# B&R Automation Studio project NAINV104C00R8L515F00 (part 6)

#### fHermesFormBoardAvailable.st
```iecst
(* Hermes Form Board Available Table Data (Total Index Written In Table) *)
FUNCTION fHermesFormBoardAvailable

	memset(ADR(pa_tyXMLTable) , 0 , SIZEOF(pa_tyXMLTable));
	iTotalIdxWrite	:= 0;

	fHermesGetTimestamp(ADR(sTimestamp) , tyDTStructure);

	pa_tyXMLTable[iTotalIdxWrite].sTitle	:= 'ST';
	pa_tyXMLTable[iTotalIdxWrite].sValue	:= 'Hermes';
	pa_tyXMLTable[iTotalIdxWrite].uiSize	:= LEN(pa_tyXMLTable[iTotalIdxWrite].sValue);

	iTotalIdxWrite	:= iTotalIdxWrite + 1;

	pa_tyXMLTable[iTotalIdxWrite].sTitle	:= 'AT';
	pa_tyXMLTable[iTotalIdxWrite].sValue	:= 'Timestamp';
	pa_tyXMLTable[iTotalIdxWrite].uiSize	:= LEN(pa_tyXMLTable[iTotalIdxWrite].sValue);

	iTotalIdxWrite	:= iTotalIdxWrite + 1;

	pa_tyXMLTable[iTotalIdxWrite].sTitle	:= 'AV';
	pa_tyXMLTable[iTotalIdxWrite].sValue	:= sTimestamp;
	pa_tyXMLTable[iTotalIdxWrite].uiSize	:= LEN(pa_tyXMLTable[iTotalIdxWrite].sValue);

	iTotalIdxWrite	:= iTotalIdxWrite + 1;

	pa_tyXMLTable[iTotalIdxWrite].sTitle	:= 'EN';
	pa_tyXMLTable[iTotalIdxWrite].sValue	:= '';
	pa_tyXMLTable[iTotalIdxWrite].uiSize	:= LEN(pa_tyXMLTable[iTotalIdxWrite].sValue);

	iTotalIdxWrite	:= iTotalIdxWrite + 1;

	pa_tyXMLTable[iTotalIdxWrite].sTitle	:= 'ST';
	pa_tyXMLTable[iTotalIdxWrite].sValue	:= 'BoardAvailable';
	pa_tyXMLTable[iTotalIdxWrite].uiSize	:= LEN(pa_tyXMLTable[iTotalIdxWrite].sValue);

	iTotalIdxWrite	:= iTotalIdxWrite + 1;

	IF tyParameter.tyAvl.bBoardId = TRUE THEN
		pa_tyXMLTable[iTotalIdxWrite].sTitle	:= 'AT';
		pa_tyXMLTable[iTotalIdxWrite].sValue	:= 'BoardId';
		pa_tyXMLTable[iTotalIdxWrite].uiSize	:= LEN(pa_tyXMLTable[iTotalIdxWrite].sValue);

		iTotalIdxWrite	:= iTotalIdxWrite + 1;

		pa_tyXMLTable[iTotalIdxWrite].sTitle	:= 'AV';
		pa_tyXMLTable[iTotalIdxWrite].sValue	:= tyParameter.tyData.sBoardId;
		pa_tyXMLTable[iTotalIdxWrite].uiSize	:= LEN(pa_tyXMLTable[iTotalIdxWrite].sValue);

		iTotalIdxWrite	:= iTotalIdxWrite + 1;
	END_IF

	IF tyParameter.tyAvl.bBoardIdCreatedBy = TRUE THEN
		pa_tyXMLTable[iTotalIdxWrite].sTitle	:= 'AT';
		pa_tyXMLTable[iTotalIdxWrite].sValue	:= 'BoardIdCreatedBy';
		pa_tyXMLTable[iTotalIdxWrite].uiSize	:= LEN(pa_tyXMLTable[iTotalIdxWrite].sValue);

		iTotalIdxWrite	:= iTotalIdxWrite + 1;

		pa_tyXMLTable[iTotalIdxWrite].sTitle	:= 'AV';
		pa_tyXMLTable[iTotalIdxWrite].sValue	:= tyParameter.tyData.sBoardIdCreatedBy;
		pa_tyXMLTable[iTotalIdxWrite].uiSize	:= LEN(pa_tyXMLTable[iTotalIdxWrite].sValue);

		iTotalIdxWrite	:= iTotalIdxWrite + 1;
	END_IF

	IF tyParameter.tyAvl.bFailedBoard = TRUE THEN
		pa_tyXMLTable[iTotalIdxWrite].sTitle	:= 'AT';
		pa_tyXMLTable[iTotalIdxWrite].sValue	:= 'FailedBoard';
		pa_tyXMLTable[iTotalIdxWrite].uiSize	:= LEN(pa_tyXMLTable[iTotalIdxWrite].sValue);

		iTotalIdxWrite	:= iTotalIdxWrite + 1;

		pa_tyXMLTable[iTotalIdxWrite].sTitle	:= 'AV';
		pa_tyXMLTable[iTotalIdxWrite].sValue	:= DINT_TO_STRING(UDINT_TO_DINT(tyParameter.tyData.eFailedBoard));
		pa_tyXMLTable[iTotalIdxWrite].uiSize	:= LEN(pa_tyXMLTable[iTotalIdxWrite].sValue);

		iTotalIdxWrite	:= iTotalIdxWrite + 1;
	END_IF

	IF tyParameter.tyAvl.bProductTypeId = TRUE THEN
		pa_tyXMLTable[iTotalIdxWrite].sTitle	:= 'AT';
		pa_tyXMLTable[iTotalIdxWrite].sValue	:= 'ProductTypeId';
		pa_tyXMLTable[iTotalIdxWrite].uiSize	:= LEN(pa_tyXMLTable[iTotalIdxWrite].sValue);

		iTotalIdxWrite	:= iTotalIdxWrite + 1;

		pa_tyXMLTable[iTotalIdxWrite].sTitle	:= 'AV';
		pa_tyXMLTable[iTotalIdxWrite].sValue	:= tyParameter.tyData.sProductTypeId;
		pa_tyXMLTable[iTotalIdxWrite].uiSize	:= LEN(pa_tyXMLTable[iTotalIdxWrite].sValue);

		iTotalIdxWrite	:= iTotalIdxWrite + 1;
	END_IF

	IF tyParameter.tyAvl.bFlippedBoard = TRUE THEN
		pa_tyXMLTable[iTotalIdxWrite].sTitle	:= 'AT';
		pa_tyXMLTable[iTotalIdxWrite].sValue	:= 'FlippedBoard';
		pa_tyXMLTable[iTotalIdxWrite].uiSize	:= LEN(pa_tyXMLTable[iTotalIdxWrite].sValue);

		iTotalIdxWrite	:= iTotalIdxWrite + 1;

		pa_tyXMLTable[iTotalIdxWrite].sTitle	:= 'AV';
		pa_tyXMLTable[iTotalIdxWrite].sValue	:= DINT_TO_STRING(UDINT_TO_DINT(tyParameter.tyData.eFlippedBoard));
		pa_tyXMLTable[iTotalIdxWrite].uiSize	:= LEN(pa_tyXMLTable[iTotalIdxWrite].sValue);

		iTotalIdxWrite	:= iTotalIdxWrite + 1;
	END_IF

	IF tyParameter.tyAvl.bTopBarcode = TRUE THEN
		pa_tyXMLTable[iTotalIdxWrite].sTitle	:= 'AT';
		pa_tyXMLTable[iTotalIdxWrite].sValue	:= 'TopBarcode';
		pa_tyXMLTable[iTotalIdxWrite].uiSize	:= LEN(pa_tyXMLTable[iTotalIdxWrite].sValue);

		iTotalIdxWrite	:= iTotalIdxWrite + 1;

		pa_tyXMLTable[iTotalIdxWrite].sTitle	:= 'AV';
		pa_tyXMLTable[iTotalIdxWrite].sValue	:= tyParameter.tyData.sTopBarcode;
		pa_tyXMLTable[iTotalIdxWrite].uiSize	:= LEN(pa_tyXMLTable[iTotalIdxWrite].sValue);

		iTotalIdxWrite	:= iTotalIdxWrite + 1;
	END_IF

	IF tyParameter.tyAvl.bBottomBarcode = TRUE THEN
		pa_tyXMLTable[iTotalIdxWrite].sTitle	:= 'AT';
		pa_tyXMLTable[iTotalIdxWrite].sValue	:= 'BottomBarcode';
		pa_tyXMLTable[iTotalIdxWrite].uiSize	:= LEN(pa_tyXMLTable[iTotalIdxWrite].sValue);

		iTotalIdxWrite	:= iTotalIdxWrite + 1;

		pa_tyXMLTable[iTotalIdxWrite].sTitle	:= 'AV';
		pa_tyXMLTable[iTotalIdxWrite].sValue	:= tyParameter.tyData.sBottomBarcode;
		pa_tyXMLTable[iTotalIdxWrite].uiSize	:= LEN(pa_tyXMLTable[iTotalIdxWrite].sValue);

		iTotalIdxWrite	:= iTotalIdxWrite + 1;
	END_IF

	IF tyParameter.tyAvl.bLength = TRUE THEN
		pa_tyXMLTable[iTotalIdxWrite].sTitle	:= 'AT';
		pa_tyXMLTable[iTotalIdxWrite].sValue	:= 'Length';
		pa_tyXMLTable[iTotalIdxWrite].uiSize	:= LEN(pa_tyXMLTable[iTotalIdxWrite].sValue);

		iTotalIdxWrite	:= iTotalIdxWrite + 1;

		pa_tyXMLTable[iTotalIdxWrite].sTitle	:= 'AV';
		pa_tyXMLTable[iTotalIdxWrite].sValue	:= REAL_TO_STRING(tyParameter.tyData.rLength);
		pa_tyXMLTable[iTotalIdxWrite].uiSize	:= LEN(pa_tyXMLTable[iTotalIdxWrite].sValue);

		iTotalIdxWrite	:= iTotalIdxWrite + 1;
	END_IF

	IF tyParameter.tyAvl.bWidth = TRUE THEN
		pa_tyXMLTable[iTotalIdxWrite].sTitle	:= 'AT';
		pa_tyXMLTable[iTotalIdxWrite].sValue	:= 'Width';
		pa_tyXMLTable[iTotalIdxWrite].uiSize	:= LEN(pa_tyXMLTable[iTotalIdxWrite].sValue);

		iTotalIdxWrite	:= iTotalIdxWrite + 1;

		pa_tyXMLTable[iTotalIdxWrite].sTitle	:= 'AV';
		pa_tyXMLTable[iTotalIdxWrite].sValue	:= REAL_TO_STRING(tyParameter.tyData.rWidth);
		pa_tyXMLTable[iTotalIdxWrite].uiSize	:= LEN(pa_tyXMLTable[iTotalIdxWrite].sValue);

		iTotalIdxWrite	:= iTotalIdxWrite + 1;
	END_IF

	IF tyParameter.tyAvl.bThickness = TRUE THEN
		pa_tyXMLTable[iTotalIdxWrite].sTitle	:= 'AT';
		pa_tyXMLTable[iTotalIdxWrite].sValue	:= 'Thickness';
		pa_tyXMLTable[iTotalIdxWrite].uiSize	:= LEN(pa_tyXMLTable[iTotalIdxWrite].sValue);

		iTotalIdxWrite	:= iTotalIdxWrite + 1;

		pa_tyXMLTable[iTotalIdxWrite].sTitle	:= 'AV';
		pa_tyXMLTable[iTotalIdxWrite].sValue	:= REAL_TO_STRING(tyParameter.tyData.rThickness);
		pa_tyXMLTable[iTotalIdxWrite].uiSize	:= LEN(pa_tyXMLTable[iTotalIdxWrite].sValue);

		iTotalIdxWrite	:= iTotalIdxWrite + 1;
	END_IF

	IF tyParameter.tyAvl.bConveyorSpeed = TRUE THEN
		pa_tyXMLTable[iTotalIdxWrite].sTitle	:= 'AT';
		pa_tyXMLTable[iTotalIdxWrite].sValue	:= 'ConveyorSpeed';
		pa_tyXMLTable[iTotalIdxWrite].uiSize	:= LEN(pa_tyXMLTable[iTotalIdxWrite].sValue);

		iTotalIdxWrite	:= iTotalIdxWrite + 1;

		pa_tyXMLTable[iTotalIdxWrite].sTitle	:= 'AV';
		pa_tyXMLTable[iTotalIdxWrite].sValue	:= REAL_TO_STRING(tyParameter.tyData.rConveyorSpeed);
		pa_tyXMLTable[iTotalIdxWrite].uiSize	:= LEN(pa_tyXMLTable[iTotalIdxWrite].sValue);

		iTotalIdxWrite	:= iTotalIdxWrite + 1;
	END_IF

	IF tyParameter.tyAvl.bTopClearanceHeight = TRUE THEN
		pa_tyXMLTable[iTotalIdxWrite].sTitle	:= 'AT';
		pa_tyXMLTable[iTotalIdxWrite].sValue	:= 'TopClearanceHeight';
		pa_tyXMLTable[iTotalIdxWrite].uiSize	:= LEN(pa_tyXMLTable[iTotalIdxWrite].sValue);

		iTotalIdxWrite	:= iTotalIdxWrite + 1;

		pa_tyXMLTable[iTotalIdxWrite].sTitle	:= 'AV';
		pa_tyXMLTable[iTotalIdxWrite].sValue	:= REAL_TO_STRING(tyParameter.tyData.rTopClearanceHeight);
		pa_tyXMLTable[iTotalIdxWrite].uiSize	:= LEN(pa_tyXMLTable[iTotalIdxWrite].sValue);

		iTotalIdxWrite	:= iTotalIdxWrite + 1;
	END_IF

	IF tyParameter.tyAvl.bBottomClearanceHeight = TRUE THEN
		pa_tyXMLTable[iTotalIdxWrite].sTitle	:= 'AT';
		pa_tyXMLTable[iTotalIdxWrite].sValue	:= 'BottomClearanceHeight';
		pa_tyXMLTable[iTotalIdxWrite].uiSize	:= LEN(pa_tyXMLTable[iTotalIdxWrite].sValue);

		iTotalIdxWrite	:= iTotalIdxWrite + 1;

		pa_tyXMLTable[iTotalIdxWrite].sTitle	:= 'AV';
		pa_tyXMLTable[iTotalIdxWrite].sValue	:= REAL_TO_STRING(tyParameter.tyData.rBottomClearanceHeight);
		pa_tyXMLTable[iTotalIdxWrite].uiSize	:= LEN(pa_tyXMLTable[iTotalIdxWrite].sValue);

		iTotalIdxWrite	:= iTotalIdxWrite + 1;
	END_IF

	IF tyParameter.tyAvl.bWeight = TRUE THEN
		pa_tyXMLTable[iTotalIdxWrite].sTitle	:= 'AT';
		pa_tyXMLTable[iTotalIdxWrite].sValue	:= 'Weight';
		pa_tyXMLTable[iTotalIdxWrite].uiSize	:= LEN(pa_tyXMLTable[iTotalIdxWrite].sValue);

		iTotalIdxWrite	:= iTotalIdxWrite + 1;

		pa_tyXMLTable[iTotalIdxWrite].sTitle	:= 'AV';
		pa_tyXMLTable[iTotalIdxWrite].sValue	:= REAL_TO_STRING(tyParameter.tyData.rWeight);
		pa_tyXMLTable[iTotalIdxWrite].uiSize	:= LEN(pa_tyXMLTable[iTotalIdxWrite].sValue);

		iTotalIdxWrite	:= iTotalIdxWrite + 1;
	END_IF

	IF tyParameter.tyAvl.bWorkOrderId = TRUE THEN
		pa_tyXMLTable[iTotalIdxWrite].sTitle	:= 'AT';
		pa_tyXMLTable[iTotalIdxWrite].sValue	:= 'WorkOrderId';
		pa_tyXMLTable[iTotalIdxWrite].uiSize	:= LEN(pa_tyXMLTable[iTotalIdxWrite].sValue);

		iTotalIdxWrite	:= iTotalIdxWrite + 1;

		pa_tyXMLTable[iTotalIdxWrite].sTitle	:= 'AV';
		pa_tyXMLTable[iTotalIdxWrite].sValue	:= tyParameter.tyData.sWorkOrderId;
		pa_tyXMLTable[iTotalIdxWrite].uiSize	:= LEN(pa_tyXMLTable[iTotalIdxWrite].sValue);

		iTotalIdxWrite	:= iTotalIdxWrite + 1;
	END_IF

	IF tyParameter.tyAvl.bBatchId = TRUE THEN
		pa_tyXMLTable[iTotalIdxWrite].sTitle	:= 'AT';
		pa_tyXMLTable[iTotalIdxWrite].sValue	:= 'BatchId';
		pa_tyXMLTable[iTotalIdxWrite].uiSize	:= LEN(pa_tyXMLTable[iTotalIdxWrite].sValue);

		iTotalIdxWrite	:= iTotalIdxWrite + 1;

		pa_tyXMLTable[iTotalIdxWrite].sTitle	:= 'AV';
		pa_tyXMLTable[iTotalIdxWrite].sValue	:= tyParameter.tyData.sBatchId;
		pa_tyXMLTable[iTotalIdxWrite].uiSize	:= LEN(pa_tyXMLTable[iTotalIdxWrite].sValue);

		iTotalIdxWrite	:= iTotalIdxWrite + 1;
	END_IF

	IF tyParameter.tyAvl.bRoute = TRUE THEN
		pa_tyXMLTable[iTotalIdxWrite].sTitle	:= 'AT';
		pa_tyXMLTable[iTotalIdxWrite].sValue	:= 'Route';
		pa_tyXMLTable[iTotalIdxWrite].uiSize	:= LEN(pa_tyXMLTable[iTotalIdxWrite].sValue);

		iTotalIdxWrite	:= iTotalIdxWrite + 1;

		pa_tyXMLTable[iTotalIdxWrite].sTitle	:= 'AV';
		pa_tyXMLTable[iTotalIdxWrite].sValue	:= INT_TO_STRING(tyParameter.tyData.iRoute);
		pa_tyXMLTable[iTotalIdxWrite].uiSize	:= LEN(pa_tyXMLTable[iTotalIdxWrite].sValue);

		iTotalIdxWrite	:= iTotalIdxWrite + 1;
	END_IF

	IF tyParameter.tyAvl.bAction = TRUE THEN
		pa_tyXMLTable[iTotalIdxWrite].sTitle	:= 'AT';
		pa_tyXMLTable[iTotalIdxWrite].sValue	:= 'Action';
		pa_tyXMLTable[iTotalIdxWrite].uiSize	:= LEN(pa_tyXMLTable[iTotalIdxWrite].sValue);

		iTotalIdxWrite	:= iTotalIdxWrite + 1;

		pa_tyXMLTable[iTotalIdxWrite].sTitle	:= 'AV';
		pa_tyXMLTable[iTotalIdxWrite].sValue	:= INT_TO_STRING(tyParameter.tyData.iAction);
		pa_tyXMLTable[iTotalIdxWrite].uiSize	:= LEN(pa_tyXMLTable[iTotalIdxWrite].sValue);

		iTotalIdxWrite	:= iTotalIdxWrite + 1;
	END_IF

	//start adding subboard
	IF tyParameter.tyAvl.tySubBoards.bSubBoardsPos[usiSubBoardCntr] <> FALSE OR
		tyParameter.tyAvl.tySubBoards.bSubBoardsBc[usiSubBoardCntr] <> FALSE OR
		tyParameter.tyAvl.tySubBoards.bSubBoardsSt[usiSubBoardCntr] <> FALSE
		THEN
		pa_tyXMLTable[iTotalIdxWrite].sTitle	:= 'EN';
		pa_tyXMLTable[iTotalIdxWrite].sValue	:= '';
		pa_tyXMLTable[iTotalIdxWrite].uiSize	:= LEN(pa_tyXMLTable[iTotalIdxWrite].sValue);

		iTotalIdxWrite	:= iTotalIdxWrite + 1;

		pa_tyXMLTable[iTotalIdxWrite].sTitle	:= 'ST';
		pa_tyXMLTable[iTotalIdxWrite].sValue	:= 'SubBoards';
		pa_tyXMLTable[iTotalIdxWrite].uiSize	:= LEN(pa_tyXMLTable[iTotalIdxWrite].sValue);

		iTotalIdxWrite	:= iTotalIdxWrite + 1;

		pa_tyXMLTable[iTotalIdxWrite].sTitle	:= 'EN';
		pa_tyXMLTable[iTotalIdxWrite].sValue	:= '';
		pa_tyXMLTable[iTotalIdxWrite].uiSize	:= LEN(pa_tyXMLTable[iTotalIdxWrite].sValue);

		iTotalIdxWrite	:= iTotalIdxWrite + 1;

		FOR usiSubBoardCntr := 0  TO SIZEOF(tyParameter.tyAvl.tySubBoards.bSubBoardsPos)/SIZEOF(tyParameter.tyAvl.tySubBoards.bSubBoardsPos[1]) -1 DO
			IF tyParameter.tyAvl.tySubBoards.bSubBoardsPos[usiSubBoardCntr] <> FALSE OR
				tyParameter.tyAvl.tySubBoards.bSubBoardsBc[usiSubBoardCntr] <> FALSE OR
				tyParameter.tyAvl.tySubBoards.bSubBoardsSt[usiSubBoardCntr] <> FALSE
				THEN
				pa_tyXMLTable[iTotalIdxWrite].sTitle	:= 'ST';
				pa_tyXMLTable[iTotalIdxWrite].sValue	:= 'SB';
				pa_tyXMLTable[iTotalIdxWrite].uiSize	:= LEN(pa_tyXMLTable[iTotalIdxWrite].sValue);

				iTotalIdxWrite	:= iTotalIdxWrite + 1;

				pa_tyXMLTable[iTotalIdxWrite].sTitle	:= 'AT';
				pa_tyXMLTable[iTotalIdxWrite].sValue	:= 'Pos';
				pa_tyXMLTable[iTotalIdxWrite].uiSize	:= LEN(pa_tyXMLTable[iTotalIdxWrite].sValue);

				iTotalIdxWrite	:= iTotalIdxWrite + 1;

				pa_tyXMLTable[iTotalIdxWrite].sTitle	:= 'AV';
				pa_tyXMLTable[iTotalIdxWrite].uiSize	:= LEN(pa_tyXMLTable[iTotalIdxWrite].sValue);
				IF tyParameter.tyAvl.tySubBoards.bSubBoardsPos[usiSubBoardCntr] <> FALSE THEN
					pa_tyXMLTable[iTotalIdxWrite].sValue	:= INT_TO_STRING(tyParameter.tyData.tySubBoards.iSubBoardsPos[usiSubBoardCntr]);
				END_IF
				iTotalIdxWrite	:= iTotalIdxWrite + 1;

				pa_tyXMLTable[iTotalIdxWrite].sTitle	:= 'AT';
				pa_tyXMLTable[iTotalIdxWrite].sValue	:= 'Bc';
				pa_tyXMLTable[iTotalIdxWrite].uiSize	:= LEN(pa_tyXMLTable[iTotalIdxWrite].sValue);

				iTotalIdxWrite	:= iTotalIdxWrite + 1;

				pa_tyXMLTable[iTotalIdxWrite].sTitle	:= 'AV';
				IF tyParameter.tyAvl.tySubBoards.bSubBoardsBc[usiSubBoardCntr] <> FALSE THEN
					pa_tyXMLTable[iTotalIdxWrite].sValue	:= tyParameter.tyData.tySubBoards.sSubBoardsBc[usiSubBoardCntr];
				END_IF
				pa_tyXMLTable[iTotalIdxWrite].uiSize	:= LEN(pa_tyXMLTable[iTotalIdxWrite].sValue);

				iTotalIdxWrite	:= iTotalIdxWrite + 1;

				pa_tyXMLTable[iTotalIdxWrite].sTitle	:= 'AT';
				pa_tyXMLTable[iTotalIdxWrite].sValue	:= 'St';
				pa_tyXMLTable[iTotalIdxWrite].uiSize	:= LEN(pa_tyXMLTable[iTotalIdxWrite].sValue);

				iTotalIdxWrite	:= iTotalIdxWrite + 1;

				pa_tyXMLTable[iTotalIdxWrite].sTitle	:= 'AV';
				IF tyParameter.tyAvl.tySubBoards.bSubBoardsSt[usiSubBoardCntr] <> FALSE THEN
					pa_tyXMLTable[iTotalIdxWrite].sValue	:= INT_TO_STRING(tyParameter.tyData.tySubBoards.iSubBoardsSt[usiSubBoardCntr]);
				END_IF
				pa_tyXMLTable[iTotalIdxWrite].uiSize	:= LEN(pa_tyXMLTable[iTotalIdxWrite].sValue);

				iTotalIdxWrite	:= iTotalIdxWrite + 1;

				pa_tyXMLTable[iTotalIdxWrite].sTitle	:= 'ES';
				pa_tyXMLTable[iTotalIdxWrite].sValue	:= '';
				pa_tyXMLTable[iTotalIdxWrite].uiSize	:= LEN(pa_tyXMLTable[iTotalIdxWrite].sValue);

				iTotalIdxWrite	:= iTotalIdxWrite + 1;
			END_IF
		END_FOR
		pa_tyXMLTable[iTotalIdxWrite].sTitle	:= 'ET';
		pa_tyXMLTable[iTotalIdxWrite].sValue	:= 'SubBoards';
		pa_tyXMLTable[iTotalIdxWrite].uiSize	:= LEN(pa_tyXMLTable[iTotalIdxWrite].sValue);

		iTotalIdxWrite	:= iTotalIdxWrite + 1;

		pa_tyXMLTable[iTotalIdxWrite].sTitle	:= 'EN';
		pa_tyXMLTable[iTotalIdxWrite].sValue	:= '';
		pa_tyXMLTable[iTotalIdxWrite].uiSize	:= LEN(pa_tyXMLTable[iTotalIdxWrite].sValue);

		iTotalIdxWrite	:= iTotalIdxWrite + 1;

		pa_tyXMLTable[iTotalIdxWrite].sTitle	:= 'ET';
		pa_tyXMLTable[iTotalIdxWrite].sValue	:= 'BoardAvailable';
		pa_tyXMLTable[iTotalIdxWrite].uiSize	:= LEN(pa_tyXMLTable[iTotalIdxWrite].sValue);

		iTotalIdxWrite	:= iTotalIdxWrite + 1;

		pa_tyXMLTable[iTotalIdxWrite].sTitle	:= 'EN';
		pa_tyXMLTable[iTotalIdxWrite].sValue	:= '';
		pa_tyXMLTable[iTotalIdxWrite].uiSize	:= LEN(pa_tyXMLTable[iTotalIdxWrite].sValue);

		iTotalIdxWrite	:= iTotalIdxWrite + 1;

	ELSE
		pa_tyXMLTable[iTotalIdxWrite].sTitle	:= 'ES';
		pa_tyXMLTable[iTotalIdxWrite].sValue	:= '';
		pa_tyXMLTable[iTotalIdxWrite].uiSize	:= LEN(pa_tyXMLTable[iTotalIdxWrite].sValue);

		iTotalIdxWrite	:= iTotalIdxWrite + 1;

	END_IF
	//to add

	pa_tyXMLTable[iTotalIdxWrite].sTitle	:= 'ET';
	pa_tyXMLTable[iTotalIdxWrite].sValue	:= 'Hermes';
	pa_tyXMLTable[iTotalIdxWrite].uiSize	:= LEN(pa_tyXMLTable[iTotalIdxWrite].sValue);

	iTotalIdxWrite	:= iTotalIdxWrite + 1;

	pa_tyXMLTable[iTotalIdxWrite].sTitle	:= 'EN';
	pa_tyXMLTable[iTotalIdxWrite].sValue	:= '';
	pa_tyXMLTable[iTotalIdxWrite].uiSize	:= LEN(pa_tyXMLTable[iTotalIdxWrite].sValue);

	iTotalIdxWrite	:= iTotalIdxWrite + 1;

	iTotalIdxWrite	:= fHermesFormBoardAvailable;

END_FUNCTION
```

#### fHermesFormRevokeBoardAvailable.st
```iecst
(* Hermes Form Revoke Board Available Table Data (Total Index Written In Table) *)
FUNCTION fHermesFormRevokeBoardAvailable

	memset(ADR(pa_tyXMLTable) , 0 , SIZEOF(pa_tyXMLTable));
	iTotalIdxWrite	:= 0;

	fHermesGetTimestamp(ADR(sTimestamp) , tyDTStructure);

	pa_tyXMLTable[iTotalIdxWrite].sTitle	:= 'ST';
	pa_tyXMLTable[iTotalIdxWrite].sValue	:= 'Hermes';
	pa_tyXMLTable[iTotalIdxWrite].uiSize	:= LEN(pa_tyXMLTable[iTotalIdxWrite].sValue);

	iTotalIdxWrite	:= iTotalIdxWrite + 1;

	pa_tyXMLTable[iTotalIdxWrite].sTitle	:= 'AT';
	pa_tyXMLTable[iTotalIdxWrite].sValue	:= 'Timestamp';
	pa_tyXMLTable[iTotalIdxWrite].uiSize	:= LEN(pa_tyXMLTable[iTotalIdxWrite].sValue);

	iTotalIdxWrite	:= iTotalIdxWrite + 1;

	pa_tyXMLTable[iTotalIdxWrite].sTitle	:= 'AV';
	pa_tyXMLTable[iTotalIdxWrite].sValue	:= sTimestamp;
	pa_tyXMLTable[iTotalIdxWrite].uiSize	:= LEN(pa_tyXMLTable[iTotalIdxWrite].sValue);

	iTotalIdxWrite	:= iTotalIdxWrite + 1;

	pa_tyXMLTable[iTotalIdxWrite].sTitle	:= 'EN';
	pa_tyXMLTable[iTotalIdxWrite].sValue	:= '';
	pa_tyXMLTable[iTotalIdxWrite].uiSize	:= LEN(pa_tyXMLTable[iTotalIdxWrite].sValue);

	iTotalIdxWrite	:= iTotalIdxWrite + 1;

	pa_tyXMLTable[iTotalIdxWrite].sTitle	:= 'ST';
	pa_tyXMLTable[iTotalIdxWrite].sValue	:= 'RevokeBoardAvailable';
	pa_tyXMLTable[iTotalIdxWrite].uiSize	:= LEN(pa_tyXMLTable[iTotalIdxWrite].sValue);

	iTotalIdxWrite	:= iTotalIdxWrite + 1;

	pa_tyXMLTable[iTotalIdxWrite].sTitle	:= 'ES';
	pa_tyXMLTable[iTotalIdxWrite].sValue	:= '';
	pa_tyXMLTable[iTotalIdxWrite].uiSize	:= LEN(pa_tyXMLTable[iTotalIdxWrite].sValue);

	iTotalIdxWrite	:= iTotalIdxWrite + 1;

	pa_tyXMLTable[iTotalIdxWrite].sTitle	:= 'ET';
	pa_tyXMLTable[iTotalIdxWrite].sValue	:= 'Hermes';
	pa_tyXMLTable[iTotalIdxWrite].uiSize	:= LEN(pa_tyXMLTable[iTotalIdxWrite].sValue);

	iTotalIdxWrite	:= iTotalIdxWrite + 1;

	pa_tyXMLTable[iTotalIdxWrite].sTitle	:= 'EN';
	pa_tyXMLTable[iTotalIdxWrite].sValue	:= '';
	pa_tyXMLTable[iTotalIdxWrite].uiSize	:= LEN(pa_tyXMLTable[iTotalIdxWrite].sValue);

	iTotalIdxWrite	:= iTotalIdxWrite + 1;

	iTotalIdxWrite	:= fHermesFormRevokeBoardAvailable;

END_FUNCTION
```

#### fHermesFormMachineReady.st
```iecst
(* Hermes Form Machine Ready Table Data (Total Index Written In Table) *)
FUNCTION fHermesFormMachineReady

	memset(ADR(pa_tyXMLTable) , 0 , SIZEOF(pa_tyXMLTable));
	iTotalIdxWrite	:= 0;

	fHermesGetTimestamp(ADR(sTimestamp) , tyDTStructure);

	pa_tyXMLTable[iTotalIdxWrite].sTitle	:= 'ST';
	pa_tyXMLTable[iTotalIdxWrite].sValue	:= 'Hermes';
	pa_tyXMLTable[iTotalIdxWrite].uiSize	:= LEN(pa_tyXMLTable[iTotalIdxWrite].sValue);

	iTotalIdxWrite	:= iTotalIdxWrite + 1;

	pa_tyXMLTable[iTotalIdxWrite].sTitle	:= 'AT';
	pa_tyXMLTable[iTotalIdxWrite].sValue	:= 'Timestamp';
	pa_tyXMLTable[iTotalIdxWrite].uiSize	:= LEN(pa_tyXMLTable[iTotalIdxWrite].sValue);

	iTotalIdxWrite	:= iTotalIdxWrite + 1;

	pa_tyXMLTable[iTotalIdxWrite].sTitle	:= 'AV';
	pa_tyXMLTable[iTotalIdxWrite].sValue	:= sTimestamp;
	pa_tyXMLTable[iTotalIdxWrite].uiSize	:= LEN(pa_tyXMLTable[iTotalIdxWrite].sValue);

	iTotalIdxWrite	:= iTotalIdxWrite + 1;

	pa_tyXMLTable[iTotalIdxWrite].sTitle	:= 'EN';
	pa_tyXMLTable[iTotalIdxWrite].sValue	:= '';
	pa_tyXMLTable[iTotalIdxWrite].uiSize	:= LEN(pa_tyXMLTable[iTotalIdxWrite].sValue);

	iTotalIdxWrite	:= iTotalIdxWrite + 1;

	pa_tyXMLTable[iTotalIdxWrite].sTitle	:= 'ST';
	pa_tyXMLTable[iTotalIdxWrite].sValue	:= 'MachineReady';
	pa_tyXMLTable[iTotalIdxWrite].uiSize	:= LEN(pa_tyXMLTable[iTotalIdxWrite].sValue);

	iTotalIdxWrite	:= iTotalIdxWrite + 1;

	IF tyParameter.tyAvl.bFailedBoard = TRUE THEN
		pa_tyXMLTable[iTotalIdxWrite].sTitle	:= 'AT';
		pa_tyXMLTable[iTotalIdxWrite].sValue	:= 'FailedBoard';
		pa_tyXMLTable[iTotalIdxWrite].uiSize	:= LEN(pa_tyXMLTable[iTotalIdxWrite].sValue);

		iTotalIdxWrite	:= iTotalIdxWrite + 1;

		pa_tyXMLTable[iTotalIdxWrite].sTitle	:= 'AV';
		pa_tyXMLTable[iTotalIdxWrite].sValue	:= DINT_TO_STRING(UDINT_TO_DINT(tyParameter.tyData.eFailedBoard));
		pa_tyXMLTable[iTotalIdxWrite].uiSize	:= LEN(pa_tyXMLTable[iTotalIdxWrite].sValue);

		iTotalIdxWrite	:= iTotalIdxWrite + 1;
	END_IF

	IF tyParameter.tyAvl.bForecastId = TRUE THEN
		pa_tyXMLTable[iTotalIdxWrite].sTitle	:= 'AT';
		pa_tyXMLTable[iTotalIdxWrite].sValue	:= 'ForecastId';
		pa_tyXMLTable[iTotalIdxWrite].uiSize	:= LEN(pa_tyXMLTable[iTotalIdxWrite].sValue);

		iTotalIdxWrite	:= iTotalIdxWrite + 1;

		pa_tyXMLTable[iTotalIdxWrite].sTitle	:= 'AV';
		pa_tyXMLTable[iTotalIdxWrite].sValue	:= tyParameter.tyData.sForecastId;
		pa_tyXMLTable[iTotalIdxWrite].uiSize	:= LEN(pa_tyXMLTable[iTotalIdxWrite].sValue);

		iTotalIdxWrite	:= iTotalIdxWrite + 1;
	END_IF

	IF tyParameter.tyAvl.bBoardId = TRUE THEN
		pa_tyXMLTable[iTotalIdxWrite].sTitle	:= 'AT';
		pa_tyXMLTable[iTotalIdxWrite].sValue	:= 'BoardId';
		pa_tyXMLTable[iTotalIdxWrite].uiSize	:= LEN(pa_tyXMLTable[iTotalIdxWrite].sValue);

		iTotalIdxWrite	:= iTotalIdxWrite + 1;

		pa_tyXMLTable[iTotalIdxWrite].sTitle	:= 'AV';
		pa_tyXMLTable[iTotalIdxWrite].sValue	:= tyParameter.tyData.sBoardId;
		pa_tyXMLTable[iTotalIdxWrite].uiSize	:= LEN(pa_tyXMLTable[iTotalIdxWrite].sValue);

		iTotalIdxWrite	:= iTotalIdxWrite + 1;
	END_IF

	IF tyParameter.tyAvl.bProductTypeId = TRUE THEN
		pa_tyXMLTable[iTotalIdxWrite].sTitle	:= 'AT';
		pa_tyXMLTable[iTotalIdxWrite].sValue	:= 'ProductTypeId';
		pa_tyXMLTable[iTotalIdxWrite].uiSize	:= LEN(pa_tyXMLTable[iTotalIdxWrite].sValue);

		iTotalIdxWrite	:= iTotalIdxWrite + 1;

		pa_tyXMLTable[iTotalIdxWrite].sTitle	:= 'AV';
		pa_tyXMLTable[iTotalIdxWrite].sValue	:= tyParameter.tyData.sProductTypeId;
		pa_tyXMLTable[iTotalIdxWrite].uiSize	:= LEN(pa_tyXMLTable[iTotalIdxWrite].sValue);

		iTotalIdxWrite	:= iTotalIdxWrite + 1;
	END_IF

	IF tyParameter.tyAvl.bFlippedBoard = TRUE THEN
		pa_tyXMLTable[iTotalIdxWrite].sTitle	:= 'AT';
		pa_tyXMLTable[iTotalIdxWrite].sValue	:= 'FlippedBoard';
		pa_tyXMLTable[iTotalIdxWrite].uiSize	:= LEN(pa_tyXMLTable[iTotalIdxWrite].sValue);

		iTotalIdxWrite	:= iTotalIdxWrite + 1;

		pa_tyXMLTable[iTotalIdxWrite].sTitle	:= 'AV';
		pa_tyXMLTable[iTotalIdxWrite].sValue	:= DINT_TO_STRING(UDINT_TO_DINT(tyParameter.tyData.eFlippedBoard));
		pa_tyXMLTable[iTotalIdxWrite].uiSize	:= LEN(pa_tyXMLTable[iTotalIdxWrite].sValue);

		iTotalIdxWrite	:= iTotalIdxWrite + 1;
	END_IF

	IF tyParameter.tyAvl.bLength = TRUE THEN
		pa_tyXMLTable[iTotalIdxWrite].sTitle	:= 'AT';
		pa_tyXMLTable[iTotalIdxWrite].sValue	:= 'Length';
		pa_tyXMLTable[iTotalIdxWrite].uiSize	:= LEN(pa_tyXMLTable[iTotalIdxWrite].sValue);

		iTotalIdxWrite	:= iTotalIdxWrite + 1;

		pa_tyXMLTable[iTotalIdxWrite].sTitle	:= 'AV';
		pa_tyXMLTable[iTotalIdxWrite].sValue	:= REAL_TO_STRING(tyParameter.tyData.rLength);
		pa_tyXMLTable[iTotalIdxWrite].uiSize	:= LEN(pa_tyXMLTable[iTotalIdxWrite].sValue);

		iTotalIdxWrite	:= iTotalIdxWrite + 1;
	END_IF

	IF tyParameter.tyAvl.bWidth = TRUE THEN
		pa_tyXMLTable[iTotalIdxWrite].sTitle	:= 'AT';
		pa_tyXMLTable[iTotalIdxWrite].sValue	:= 'Width';
		pa_tyXMLTable[iTotalIdxWrite].uiSize	:= LEN(pa_tyXMLTable[iTotalIdxWrite].sValue);

		iTotalIdxWrite	:= iTotalIdxWrite + 1;

		pa_tyXMLTable[iTotalIdxWrite].sTitle	:= 'AV';
		pa_tyXMLTable[iTotalIdxWrite].sValue	:= REAL_TO_STRING(tyParameter.tyData.rWidth);
		pa_tyXMLTable[iTotalIdxWrite].uiSize	:= LEN(pa_tyXMLTable[iTotalIdxWrite].sValue);

		iTotalIdxWrite	:= iTotalIdxWrite + 1;
	END_IF

	IF tyParameter.tyAvl.bThickness = TRUE THEN
		pa_tyXMLTable[iTotalIdxWrite].sTitle	:= 'AT';
		pa_tyXMLTable[iTotalIdxWrite].sValue	:= 'Thickness';
		pa_tyXMLTable[iTotalIdxWrite].uiSize	:= LEN(pa_tyXMLTable[iTotalIdxWrite].sValue);

		iTotalIdxWrite	:= iTotalIdxWrite + 1;

		pa_tyXMLTable[iTotalIdxWrite].sTitle	:= 'AV';
		pa_tyXMLTable[iTotalIdxWrite].sValue	:= REAL_TO_STRING(tyParameter.tyData.rThickness);
		pa_tyXMLTable[iTotalIdxWrite].uiSize	:= LEN(pa_tyXMLTable[iTotalIdxWrite].sValue);

		iTotalIdxWrite	:= iTotalIdxWrite + 1;
	END_IF

	IF tyParameter.tyAvl.bConveyorSpeed = TRUE THEN
		pa_tyXMLTable[iTotalIdxWrite].sTitle	:= 'AT';
		pa_tyXMLTable[iTotalIdxWrite].sValue	:= 'ConveyorSpeed';
		pa_tyXMLTable[iTotalIdxWrite].uiSize	:= LEN(pa_tyXMLTable[iTotalIdxWrite].sValue);

		iTotalIdxWrite	:= iTotalIdxWrite + 1;

		pa_tyXMLTable[iTotalIdxWrite].sTitle	:= 'AV';
		pa_tyXMLTable[iTotalIdxWrite].sValue	:= REAL_TO_STRING(tyParameter.tyData.rConveyorSpeed);
		pa_tyXMLTable[iTotalIdxWrite].uiSize	:= LEN(pa_tyXMLTable[iTotalIdxWrite].sValue);

		iTotalIdxWrite	:= iTotalIdxWrite + 1;
	END_IF

	IF tyParameter.tyAvl.bTopClearanceHeight = TRUE THEN
		pa_tyXMLTable[iTotalIdxWrite].sTitle	:= 'AT';
		pa_tyXMLTable[iTotalIdxWrite].sValue	:= 'TopClearanceHeight';
		pa_tyXMLTable[iTotalIdxWrite].uiSize	:= LEN(pa_tyXMLTable[iTotalIdxWrite].sValue);

		iTotalIdxWrite	:= iTotalIdxWrite + 1;

		pa_tyXMLTable[iTotalIdxWrite].sTitle	:= 'AV';
		pa_tyXMLTable[iTotalIdxWrite].sValue	:= REAL_TO_STRING(tyParameter.tyData.rTopClearanceHeight);
		pa_tyXMLTable[iTotalIdxWrite].uiSize	:= LEN(pa_tyXMLTable[iTotalIdxWrite].sValue);

		iTotalIdxWrite	:= iTotalIdxWrite + 1;
	END_IF

	IF tyParameter.tyAvl.bBottomClearanceHeight = TRUE THEN
		pa_tyXMLTable[iTotalIdxWrite].sTitle	:= 'AT';
		pa_tyXMLTable[iTotalIdxWrite].sValue	:= 'BottomClearanceHeight';
		pa_tyXMLTable[iTotalIdxWrite].uiSize	:= LEN(pa_tyXMLTable[iTotalIdxWrite].sValue);

		iTotalIdxWrite	:= iTotalIdxWrite + 1;

		pa_tyXMLTable[iTotalIdxWrite].sTitle	:= 'AV';
		pa_tyXMLTable[iTotalIdxWrite].sValue	:= REAL_TO_STRING(tyParameter.tyData.rBottomClearanceHeight);
		pa_tyXMLTable[iTotalIdxWrite].uiSize	:= LEN(pa_tyXMLTable[iTotalIdxWrite].sValue);

		iTotalIdxWrite	:= iTotalIdxWrite + 1;
	END_IF

	IF tyParameter.tyAvl.bWeight = TRUE THEN
		pa_tyXMLTable[iTotalIdxWrite].sTitle	:= 'AT';
		pa_tyXMLTable[iTotalIdxWrite].sValue	:= 'Weight';
		pa_tyXMLTable[iTotalIdxWrite].uiSize	:= LEN(pa_tyXMLTable[iTotalIdxWrite].sValue);

		iTotalIdxWrite	:= iTotalIdxWrite + 1;

		pa_tyXMLTable[iTotalIdxWrite].sTitle	:= 'AV';
		pa_tyXMLTable[iTotalIdxWrite].sValue	:= REAL_TO_STRING(tyParameter.tyData.rWeight);
		pa_tyXMLTable[iTotalIdxWrite].uiSize	:= LEN(pa_tyXMLTable[iTotalIdxWrite].sValue);

		iTotalIdxWrite	:= iTotalIdxWrite + 1;
	END_IF

	IF tyParameter.tyAvl.bWorkOrderId = TRUE THEN
		pa_tyXMLTable[iTotalIdxWrite].sTitle	:= 'AT';
		pa_tyXMLTable[iTotalIdxWrite].sValue	:= 'WorkOrderId';
		pa_tyXMLTable[iTotalIdxWrite].uiSize	:= LEN(pa_tyXMLTable[iTotalIdxWrite].sValue);

		iTotalIdxWrite	:= iTotalIdxWrite + 1;

		pa_tyXMLTable[iTotalIdxWrite].sTitle	:= 'AV';
		pa_tyXMLTable[iTotalIdxWrite].sValue	:= tyParameter.tyData.sWorkOrderId;
		pa_tyXMLTable[iTotalIdxWrite].uiSize	:= LEN(pa_tyXMLTable[iTotalIdxWrite].sValue);

		iTotalIdxWrite	:= iTotalIdxWrite + 1;
	END_IF

	IF tyParameter.tyAvl.bBatchId = TRUE THEN
		pa_tyXMLTable[iTotalIdxWrite].sTitle	:= 'AT';
		pa_tyXMLTable[iTotalIdxWrite].sValue	:= 'BatchId';
		pa_tyXMLTable[iTotalIdxWrite].uiSize	:= LEN(pa_tyXMLTable[iTotalIdxWrite].sValue);

		iTotalIdxWrite	:= iTotalIdxWrite + 1;

		pa_tyXMLTable[iTotalIdxWrite].sTitle	:= 'AV';
		pa_tyXMLTable[iTotalIdxWrite].sValue	:= tyParameter.tyData.sBatchId;
		pa_tyXMLTable[iTotalIdxWrite].uiSize	:= LEN(pa_tyXMLTable[iTotalIdxWrite].sValue);

		iTotalIdxWrite	:= iTotalIdxWrite + 1;
	END_IF

	pa_tyXMLTable[iTotalIdxWrite].sTitle	:= 'ES';
	pa_tyXMLTable[iTotalIdxWrite].sValue	:= '';
	pa_tyXMLTable[iTotalIdxWrite].uiSize	:= LEN(pa_tyXMLTable[iTotalIdxWrite].sValue);

	iTotalIdxWrite	:= iTotalIdxWrite + 1;

	pa_tyXMLTable[iTotalIdxWrite].sTitle	:= 'ET';
	pa_tyXMLTable[iTotalIdxWrite].sValue	:= 'Hermes';
	pa_tyXMLTable[iTotalIdxWrite].uiSize	:= LEN(pa_tyXMLTable[iTotalIdxWrite].sValue);

	iTotalIdxWrite	:= iTotalIdxWrite + 1;

	pa_tyXMLTable[iTotalIdxWrite].sTitle	:= 'EN';
	pa_tyXMLTable[iTotalIdxWrite].sValue	:= '';
	pa_tyXMLTable[iTotalIdxWrite].uiSize	:= LEN(pa_tyXMLTable[iTotalIdxWrite].sValue);

	iTotalIdxWrite	:= iTotalIdxWrite + 1;

	iTotalIdxWrite	:= fHermesFormMachineReady;

END_FUNCTION
```

#### fHermesFormRevokeMachineReady.st
```iecst
(* Hermes Form Revoke Machine Ready Table Data (Total Index Written In Table) *)
FUNCTION fHermesFormRevokeMachineReady

	memset(ADR(pa_tyXMLTable) , 0 , SIZEOF(pa_tyXMLTable));
	iTotalIdxWrite	:= 0;

	fHermesGetTimestamp(ADR(sTimestamp) , tyDTStructure);

	pa_tyXMLTable[iTotalIdxWrite].sTitle	:= 'ST';
	pa_tyXMLTable[iTotalIdxWrite].sValue	:= 'Hermes';
	pa_tyXMLTable[iTotalIdxWrite].uiSize	:= LEN(pa_tyXMLTable[iTotalIdxWrite].sValue);

	iTotalIdxWrite	:= iTotalIdxWrite + 1;

	pa_tyXMLTable[iTotalIdxWrite].sTitle	:= 'AT';
	pa_tyXMLTable[iTotalIdxWrite].sValue	:= 'Timestamp';
	pa_tyXMLTable[iTotalIdxWrite].uiSize	:= LEN(pa_tyXMLTable[iTotalIdxWrite].sValue);

	iTotalIdxWrite	:= iTotalIdxWrite + 1;

	pa_tyXMLTable[iTotalIdxWrite].sTitle	:= 'AV';
	pa_tyXMLTable[iTotalIdxWrite].sValue	:= sTimestamp;
	pa_tyXMLTable[iTotalIdxWrite].uiSize	:= LEN(pa_tyXMLTable[iTotalIdxWrite].sValue);

	iTotalIdxWrite	:= iTotalIdxWrite + 1;

	pa_tyXMLTable[iTotalIdxWrite].sTitle	:= 'EN';
	pa_tyXMLTable[iTotalIdxWrite].sValue	:= '';
	pa_tyXMLTable[iTotalIdxWrite].uiSize	:= LEN(pa_tyXMLTable[iTotalIdxWrite].sValue);

	iTotalIdxWrite	:= iTotalIdxWrite + 1;

	pa_tyXMLTable[iTotalIdxWrite].sTitle	:= 'ST';
	pa_tyXMLTable[iTotalIdxWrite].sValue	:= 'RevokeMachineReady';
	pa_tyXMLTable[iTotalIdxWrite].uiSize	:= LEN(pa_tyXMLTable[iTotalIdxWrite].sValue);

	iTotalIdxWrite	:= iTotalIdxWrite + 1;

	pa_tyXMLTable[iTotalIdxWrite].sTitle	:= 'ES';
	pa_tyXMLTable[iTotalIdxWrite].sValue	:= '';
	pa_tyXMLTable[iTotalIdxWrite].uiSize	:= LEN(pa_tyXMLTable[iTotalIdxWrite].sValue);

	iTotalIdxWrite	:= iTotalIdxWrite + 1;

	pa_tyXMLTable[iTotalIdxWrite].sTitle	:= 'ET';
	pa_tyXMLTable[iTotalIdxWrite].sValue	:= 'Hermes';
	pa_tyXMLTable[iTotalIdxWrite].uiSize	:= LEN(pa_tyXMLTable[iTotalIdxWrite].sValue);

	iTotalIdxWrite	:= iTotalIdxWrite + 1;

	pa_tyXMLTable[iTotalIdxWrite].sTitle	:= 'EN';
	pa_tyXMLTable[iTotalIdxWrite].sValue	:= '';
	pa_tyXMLTable[iTotalIdxWrite].uiSize	:= LEN(pa_tyXMLTable[iTotalIdxWrite].sValue);

	iTotalIdxWrite	:= iTotalIdxWrite + 1;

	iTotalIdxWrite	:= fHermesFormRevokeMachineReady;

END_FUNCTION
```

#### fHermesFormStartTransport.st
```iecst
(* Hermes Form Start Transport Table Data (Total Index Written In Table) *)
FUNCTION fHermesFormStartTransport

	memset(ADR(pa_tyXMLTable) , 0 , SIZEOF(pa_tyXMLTable));
	iTotalIdxWrite	:= 0;

	fHermesGetTimestamp(ADR(sTimestamp) , tyDTStructure);

	pa_tyXMLTable[iTotalIdxWrite].sTitle	:= 'ST';
	pa_tyXMLTable[iTotalIdxWrite].sValue	:= 'Hermes';
	pa_tyXMLTable[iTotalIdxWrite].uiSize	:= LEN(pa_tyXMLTable[iTotalIdxWrite].sValue);

	iTotalIdxWrite	:= iTotalIdxWrite + 1;

	pa_tyXMLTable[iTotalIdxWrite].sTitle	:= 'AT';
	pa_tyXMLTable[iTotalIdxWrite].sValue	:= 'Timestamp';
	pa_tyXMLTable[iTotalIdxWrite].uiSize	:= LEN(pa_tyXMLTable[iTotalIdxWrite].sValue);

	iTotalIdxWrite	:= iTotalIdxWrite + 1;

	pa_tyXMLTable[iTotalIdxWrite].sTitle	:= 'AV';
	pa_tyXMLTable[iTotalIdxWrite].sValue	:= sTimestamp;
	pa_tyXMLTable[iTotalIdxWrite].uiSize	:= LEN(pa_tyXMLTable[iTotalIdxWrite].sValue);

	iTotalIdxWrite	:= iTotalIdxWrite + 1;

	pa_tyXMLTable[iTotalIdxWrite].sTitle	:= 'EN';
	pa_tyXMLTable[iTotalIdxWrite].sValue	:= '';
	pa_tyXMLTable[iTotalIdxWrite].uiSize	:= LEN(pa_tyXMLTable[iTotalIdxWrite].sValue);

	iTotalIdxWrite	:= iTotalIdxWrite + 1;

	pa_tyXMLTable[iTotalIdxWrite].sTitle	:= 'ST';
	pa_tyXMLTable[iTotalIdxWrite].sValue	:= 'StartTransport';
	pa_tyXMLTable[iTotalIdxWrite].uiSize	:= LEN(pa_tyXMLTable[iTotalIdxWrite].sValue);

	iTotalIdxWrite	:= iTotalIdxWrite + 1;

	IF tyParameter.tyAvl.bBoardId = TRUE THEN
		pa_tyXMLTable[iTotalIdxWrite].sTitle	:= 'AT';
		pa_tyXMLTable[iTotalIdxWrite].sValue	:= 'BoardId';
		pa_tyXMLTable[iTotalIdxWrite].uiSize	:= LEN(pa_tyXMLTable[iTotalIdxWrite].sValue);

		iTotalIdxWrite	:= iTotalIdxWrite + 1;

		pa_tyXMLTable[iTotalIdxWrite].sTitle	:= 'AV';
		pa_tyXMLTable[iTotalIdxWrite].sValue	:= tyParameter.tyData.sBoardId;
		pa_tyXMLTable[iTotalIdxWrite].uiSize	:= LEN(pa_tyXMLTable[iTotalIdxWrite].sValue);

		iTotalIdxWrite	:= iTotalIdxWrite + 1;
	END_IF

	IF tyParameter.tyAvl.bConveyorSpeed = TRUE THEN
		pa_tyXMLTable[iTotalIdxWrite].sTitle	:= 'AT';
		pa_tyXMLTable[iTotalIdxWrite].sValue	:= 'ConveyorSpeed';
		pa_tyXMLTable[iTotalIdxWrite].uiSize	:= LEN(pa_tyXMLTable[iTotalIdxWrite].sValue);

		iTotalIdxWrite	:= iTotalIdxWrite + 1;

		pa_tyXMLTable[iTotalIdxWrite].sTitle	:= 'AV';
		pa_tyXMLTable[iTotalIdxWrite].sValue	:= REAL_TO_STRING(tyParameter.tyData.rConveyorSpeed);
		pa_tyXMLTable[iTotalIdxWrite].uiSize	:= LEN(pa_tyXMLTable[iTotalIdxWrite].sValue);

		iTotalIdxWrite	:= iTotalIdxWrite + 1;
	END_IF

	pa_tyXMLTable[iTotalIdxWrite].sTitle	:= 'ES';
	pa_tyXMLTable[iTotalIdxWrite].sValue	:= '';
	pa_tyXMLTable[iTotalIdxWrite].uiSize	:= LEN(pa_tyXMLTable[iTotalIdxWrite].sValue);

	iTotalIdxWrite	:= iTotalIdxWrite + 1;

	pa_tyXMLTable[iTotalIdxWrite].sTitle	:= 'ET';
	pa_tyXMLTable[iTotalIdxWrite].sValue	:= 'Hermes';
	pa_tyXMLTable[iTotalIdxWrite].uiSize	:= LEN(pa_tyXMLTable[iTotalIdxWrite].sValue);

	iTotalIdxWrite	:= iTotalIdxWrite + 1;

	pa_tyXMLTable[iTotalIdxWrite].sTitle	:= 'EN';
	pa_tyXMLTable[iTotalIdxWrite].sValue	:= '';
	pa_tyXMLTable[iTotalIdxWrite].uiSize	:= LEN(pa_tyXMLTable[iTotalIdxWrite].sValue);

	iTotalIdxWrite	:= iTotalIdxWrite + 1;

	iTotalIdxWrite	:= fHermesFormStartTransport;

END_FUNCTION
```

#### fHermesFormStopTransport.st
```iecst
(* Hermes Form Stop Transport Table Data (Total Index Written In Table) *)
FUNCTION fHermesFormStopTransport

	memset(ADR(pa_tyXMLTable) , 0 , SIZEOF(pa_tyXMLTable));
	iTotalIdxWrite	:= 0;

	fHermesGetTimestamp(ADR(sTimestamp) , tyDTStructure);

	pa_tyXMLTable[iTotalIdxWrite].sTitle	:= 'ST';
	pa_tyXMLTable[iTotalIdxWrite].sValue	:= 'Hermes';
	pa_tyXMLTable[iTotalIdxWrite].uiSize	:= LEN(pa_tyXMLTable[iTotalIdxWrite].sValue);

	iTotalIdxWrite	:= iTotalIdxWrite + 1;

	pa_tyXMLTable[iTotalIdxWrite].sTitle	:= 'AT';
	pa_tyXMLTable[iTotalIdxWrite].sValue	:= 'Timestamp';
	pa_tyXMLTable[iTotalIdxWrite].uiSize	:= LEN(pa_tyXMLTable[iTotalIdxWrite].sValue);

	iTotalIdxWrite	:= iTotalIdxWrite + 1;

	pa_tyXMLTable[iTotalIdxWrite].sTitle	:= 'AV';
	pa_tyXMLTable[iTotalIdxWrite].sValue	:= sTimestamp;
	pa_tyXMLTable[iTotalIdxWrite].uiSize	:= LEN(pa_tyXMLTable[iTotalIdxWrite].sValue);

	iTotalIdxWrite	:= iTotalIdxWrite + 1;

	pa_tyXMLTable[iTotalIdxWrite].sTitle	:= 'EN';
	pa_tyXMLTable[iTotalIdxWrite].sValue	:= '';
	pa_tyXMLTable[iTotalIdxWrite].uiSize	:= LEN(pa_tyXMLTable[iTotalIdxWrite].sValue);

	iTotalIdxWrite	:= iTotalIdxWrite + 1;

	pa_tyXMLTable[iTotalIdxWrite].sTitle	:= 'ST';
	pa_tyXMLTable[iTotalIdxWrite].sValue	:= 'StopTransport';
	pa_tyXMLTable[iTotalIdxWrite].uiSize	:= LEN(pa_tyXMLTable[iTotalIdxWrite].sValue);

	iTotalIdxWrite	:= iTotalIdxWrite + 1;

	IF tyParameter.tyAvl.bTransferState = TRUE THEN
		pa_tyXMLTable[iTotalIdxWrite].sTitle	:= 'AT';
		pa_tyXMLTable[iTotalIdxWrite].sValue	:= 'TransferState';
		pa_tyXMLTable[iTotalIdxWrite].uiSize	:= LEN(pa_tyXMLTable[iTotalIdxWrite].sValue);

		iTotalIdxWrite	:= iTotalIdxWrite + 1;

		pa_tyXMLTable[iTotalIdxWrite].sTitle	:= 'AV';
		pa_tyXMLTable[iTotalIdxWrite].sValue	:= DINT_TO_STRING(UDINT_TO_DINT(tyParameter.tyData.eTransferState));
		pa_tyXMLTable[iTotalIdxWrite].uiSize	:= LEN(pa_tyXMLTable[iTotalIdxWrite].sValue);

		iTotalIdxWrite	:= iTotalIdxWrite + 1;
	END_IF

	IF tyParameter.tyAvl.bBoardId = TRUE THEN
		pa_tyXMLTable[iTotalIdxWrite].sTitle	:= 'AT';
		pa_tyXMLTable[iTotalIdxWrite].sValue	:= 'BoardId';
		pa_tyXMLTable[iTotalIdxWrite].uiSize	:= LEN(pa_tyXMLTable[iTotalIdxWrite].sValue);

		iTotalIdxWrite	:= iTotalIdxWrite + 1;

		pa_tyXMLTable[iTotalIdxWrite].sTitle	:= 'AV';
		pa_tyXMLTable[iTotalIdxWrite].sValue	:= tyParameter.tyData.sBoardId;
		pa_tyXMLTable[iTotalIdxWrite].uiSize	:= LEN(pa_tyXMLTable[iTotalIdxWrite].sValue);

		iTotalIdxWrite	:= iTotalIdxWrite + 1;
	END_IF

	pa_tyXMLTable[iTotalIdxWrite].sTitle	:= 'ES';
	pa_tyXMLTable[iTotalIdxWrite].sValue	:= '';
	pa_tyXMLTable[iTotalIdxWrite].uiSize	:= LEN(pa_tyXMLTable[iTotalIdxWrite].sValue);

	iTotalIdxWrite	:= iTotalIdxWrite + 1;

	pa_tyXMLTable[iTotalIdxWrite].sTitle	:= 'ET';
	pa_tyXMLTable[iTotalIdxWrite].sValue	:= 'Hermes';
	pa_tyXMLTable[iTotalIdxWrite].uiSize	:= LEN(pa_tyXMLTable[iTotalIdxWrite].sValue);

	iTotalIdxWrite	:= iTotalIdxWrite + 1;

	pa_tyXMLTable[iTotalIdxWrite].sTitle	:= 'EN';
	pa_tyXMLTable[iTotalIdxWrite].sValue	:= '';
	pa_tyXMLTable[iTotalIdxWrite].uiSize	:= LEN(pa_tyXMLTable[iTotalIdxWrite].sValue);

	iTotalIdxWrite	:= iTotalIdxWrite + 1;

	iTotalIdxWrite	:= fHermesFormStopTransport;

END_FUNCTION
```

#### fHermesFormTransportFinished.st
```iecst
(* Hermes Form Transport Finished Table Data (Total Index Written In Table) *)
FUNCTION fHermesFormTransportFinished

	memset(ADR(pa_tyXMLTable) , 0 , SIZEOF(pa_tyXMLTable));
	iTotalIdxWrite	:= 0;

	fHermesGetTimestamp(ADR(sTimestamp) , tyDTStructure);

	pa_tyXMLTable[iTotalIdxWrite].sTitle	:= 'ST';
	pa_tyXMLTable[iTotalIdxWrite].sValue	:= 'Hermes';
	pa_tyXMLTable[iTotalIdxWrite].uiSize	:= LEN(pa_tyXMLTable[iTotalIdxWrite].sValue);

	iTotalIdxWrite	:= iTotalIdxWrite + 1;

	pa_tyXMLTable[iTotalIdxWrite].sTitle	:= 'AT';
	pa_tyXMLTable[iTotalIdxWrite].sValue	:= 'Timestamp';
	pa_tyXMLTable[iTotalIdxWrite].uiSize	:= LEN(pa_tyXMLTable[iTotalIdxWrite].sValue);

	iTotalIdxWrite	:= iTotalIdxWrite + 1;

	pa_tyXMLTable[iTotalIdxWrite].sTitle	:= 'AV';
	pa_tyXMLTable[iTotalIdxWrite].sValue	:= sTimestamp;
	pa_tyXMLTable[iTotalIdxWrite].uiSize	:= LEN(pa_tyXMLTable[iTotalIdxWrite].sValue);

	iTotalIdxWrite	:= iTotalIdxWrite + 1;

	pa_tyXMLTable[iTotalIdxWrite].sTitle	:= 'EN';
	pa_tyXMLTable[iTotalIdxWrite].sValue	:= '';
	pa_tyXMLTable[iTotalIdxWrite].uiSize	:= LEN(pa_tyXMLTable[iTotalIdxWrite].sValue);

	iTotalIdxWrite	:= iTotalIdxWrite + 1;

	pa_tyXMLTable[iTotalIdxWrite].sTitle	:= 'ST';
	pa_tyXMLTable[iTotalIdxWrite].sValue	:= 'TransportFinished';
	pa_tyXMLTable[iTotalIdxWrite].uiSize	:= LEN(pa_tyXMLTable[iTotalIdxWrite].sValue);

	iTotalIdxWrite	:= iTotalIdxWrite + 1;

	IF tyParameter.tyAvl.bTransferState = TRUE THEN
		pa_tyXMLTable[iTotalIdxWrite].sTitle	:= 'AT';
		pa_tyXMLTable[iTotalIdxWrite].sValue	:= 'TransferState';
		pa_tyXMLTable[iTotalIdxWrite].uiSize	:= LEN(pa_tyXMLTable[iTotalIdxWrite].sValue);

		iTotalIdxWrite	:= iTotalIdxWrite + 1;

		pa_tyXMLTable[iTotalIdxWrite].sTitle	:= 'AV';
		pa_tyXMLTable[iTotalIdxWrite].sValue	:= DINT_TO_STRING(UDINT_TO_DINT(tyParameter.tyData.eTransferState));
		pa_tyXMLTable[iTotalIdxWrite].uiSize	:= LEN(pa_tyXMLTable[iTotalIdxWrite].sValue);

		iTotalIdxWrite	:= iTotalIdxWrite + 1;
	END_IF

	IF tyParameter.tyAvl.bBoardId = TRUE THEN
		pa_tyXMLTable[iTotalIdxWrite].sTitle	:= 'AT';
		pa_tyXMLTable[iTotalIdxWrite].sValue	:= 'BoardId';
		pa_tyXMLTable[iTotalIdxWrite].uiSize	:= LEN(pa_tyXMLTable[iTotalIdxWrite].sValue);

		iTotalIdxWrite	:= iTotalIdxWrite + 1;

		pa_tyXMLTable[iTotalIdxWrite].sTitle	:= 'AV';
		pa_tyXMLTable[iTotalIdxWrite].sValue	:= tyParameter.tyData.sBoardId;
		pa_tyXMLTable[iTotalIdxWrite].uiSize	:= LEN(pa_tyXMLTable[iTotalIdxWrite].sValue);

		iTotalIdxWrite	:= iTotalIdxWrite + 1;
	END_IF

	pa_tyXMLTable[iTotalIdxWrite].sTitle	:= 'ES';
	pa_tyXMLTable[iTotalIdxWrite].sValue	:= '';
	pa_tyXMLTable[iTotalIdxWrite].uiSize	:= LEN(pa_tyXMLTable[iTotalIdxWrite].sValue);

	iTotalIdxWrite	:= iTotalIdxWrite + 1;

	pa_tyXMLTable[iTotalIdxWrite].sTitle	:= 'ET';
	pa_tyXMLTable[iTotalIdxWrite].sValue	:= 'Hermes';
	pa_tyXMLTable[iTotalIdxWrite].uiSize	:= LEN(pa_tyXMLTable[iTotalIdxWrite].sValue);

	iTotalIdxWrite	:= iTotalIdxWrite + 1;

	pa_tyXMLTable[iTotalIdxWrite].sTitle	:= 'EN';
	pa_tyXMLTable[iTotalIdxWrite].sValue	:= '';
	pa_tyXMLTable[iTotalIdxWrite].uiSize	:= LEN(pa_tyXMLTable[iTotalIdxWrite].sValue);

	iTotalIdxWrite	:= iTotalIdxWrite + 1;

	iTotalIdxWrite	:= fHermesFormTransportFinished;

END_FUNCTION
```

#### fHermesFormSetConfiguration.st
```iecst
(* Hermes Form Set Configuration Table Data (Total Index Written In Table) *)
FUNCTION fHermesFormSetConfiguration

	memset(ADR(pa_tyXMLTable) , 0 , SIZEOF(pa_tyXMLTable));
	iTotalIdxWrite	:= 0;

	fHermesGetTimestamp(ADR(sTimestamp) , tyDTStructure);

	pa_tyXMLTable[iTotalIdxWrite].sTitle	:= 'ST';
	pa_tyXMLTable[iTotalIdxWrite].sValue	:= 'Hermes';
	pa_tyXMLTable[iTotalIdxWrite].uiSize	:= LEN(pa_tyXMLTable[iTotalIdxWrite].sValue);

	iTotalIdxWrite	:= iTotalIdxWrite + 1;

	pa_tyXMLTable[iTotalIdxWrite].sTitle	:= 'AT';
	pa_tyXMLTable[iTotalIdxWrite].sValue	:= 'Timestamp';
	pa_tyXMLTable[iTotalIdxWrite].uiSize	:= LEN(pa_tyXMLTable[iTotalIdxWrite].sValue);

	iTotalIdxWrite	:= iTotalIdxWrite + 1;

	pa_tyXMLTable[iTotalIdxWrite].sTitle	:= 'AV';
	pa_tyXMLTable[iTotalIdxWrite].sValue	:= sTimestamp;
	pa_tyXMLTable[iTotalIdxWrite].uiSize	:= LEN(pa_tyXMLTable[iTotalIdxWrite].sValue);

	iTotalIdxWrite	:= iTotalIdxWrite + 1;

	pa_tyXMLTable[iTotalIdxWrite].sTitle	:= 'EN';
	pa_tyXMLTable[iTotalIdxWrite].sValue	:= '';
	pa_tyXMLTable[iTotalIdxWrite].uiSize	:= LEN(pa_tyXMLTable[iTotalIdxWrite].sValue);

	iTotalIdxWrite	:= iTotalIdxWrite + 1;

	pa_tyXMLTable[iTotalIdxWrite].sTitle	:= 'ST';
	pa_tyXMLTable[iTotalIdxWrite].sValue	:= 'SetConfiguration';
	pa_tyXMLTable[iTotalIdxWrite].uiSize	:= LEN(pa_tyXMLTable[iTotalIdxWrite].sValue);

	iTotalIdxWrite	:= iTotalIdxWrite + 1;

	IF tyParameter.tyAvl.bMachineId = TRUE THEN
		pa_tyXMLTable[iTotalIdxWrite].sTitle	:= 'AT';
		pa_tyXMLTable[iTotalIdxWrite].sValue	:= 'MachineId';
		pa_tyXMLTable[iTotalIdxWrite].uiSize	:= LEN(pa_tyXMLTable[iTotalIdxWrite].sValue);

		iTotalIdxWrite	:= iTotalIdxWrite + 1;

		pa_tyXMLTable[iTotalIdxWrite].sTitle	:= 'AV';
		pa_tyXMLTable[iTotalIdxWrite].sValue	:= tyParameter.tyData.sMachineId;
		pa_tyXMLTable[iTotalIdxWrite].uiSize	:= LEN(pa_tyXMLTable[iTotalIdxWrite].sValue);

		iTotalIdxWrite	:= iTotalIdxWrite + 1;
	END_IF

	IF tyParameter.tyAvl.bSupervisorySystemPort = TRUE THEN
		pa_tyXMLTable[iTotalIdxWrite].sTitle	:= 'AT';
		pa_tyXMLTable[iTotalIdxWrite].sValue	:= 'SupervisorySystemPort';
		pa_tyXMLTable[iTotalIdxWrite].uiSize	:= LEN(pa_tyXMLTable[iTotalIdxWrite].sValue);

		iTotalIdxWrite	:= iTotalIdxWrite + 1;

		pa_tyXMLTable[iTotalIdxWrite].sTitle	:= 'AV';
		pa_tyXMLTable[iTotalIdxWrite].sValue	:= UINT_TO_STRING(tyParameter.tyData.uiSupervisorySystemPort);
		pa_tyXMLTable[iTotalIdxWrite].uiSize	:= LEN(pa_tyXMLTable[iTotalIdxWrite].sValue);

		iTotalIdxWrite	:= iTotalIdxWrite + 1;
	END_IF

	pa_tyXMLTable[iTotalIdxWrite].sTitle	:= 'EN';
	pa_tyXMLTable[iTotalIdxWrite].sValue	:= '';
	pa_tyXMLTable[iTotalIdxWrite].uiSize	:= LEN(pa_tyXMLTable[iTotalIdxWrite].sValue);

	iTotalIdxWrite	:= iTotalIdxWrite + 1;

	IF tyParameter.tyAvl.iUpstreamConfigurations > 0 THEN

		pa_tyXMLTable[iTotalIdxWrite].sTitle	:= 'ST';
		pa_tyXMLTable[iTotalIdxWrite].sValue	:= 'UpstreamConfigurations';
		pa_tyXMLTable[iTotalIdxWrite].uiSize	:= LEN(pa_tyXMLTable[iTotalIdxWrite].sValue);

		iTotalIdxWrite	:= iTotalIdxWrite + 1;

		pa_tyXMLTable[iTotalIdxWrite].sTitle	:= 'EN';
		pa_tyXMLTable[iTotalIdxWrite].sValue	:= '';
		pa_tyXMLTable[iTotalIdxWrite].uiSize	:= LEN(pa_tyXMLTable[iTotalIdxWrite].sValue);

		iTotalIdxWrite	:= iTotalIdxWrite + 1;

		IF tyParameter.tyAvl.iUpstreamConfigurations < 4 THEN
			iConfiguration	:= tyParameter.tyAvl.iUpstreamConfigurations - 1;
		ELSE
			iConfiguration	:= 2;
		END_IF

		FOR i := 0 TO iConfiguration DO

			pa_tyXMLTable[iTotalIdxWrite].sTitle	:= 'ST';
			pa_tyXMLTable[iTotalIdxWrite].sValue	:= 'UpstreamConfiguration';
			pa_tyXMLTable[iTotalIdxWrite].uiSize	:= LEN(pa_tyXMLTable[iTotalIdxWrite].sValue);

			iTotalIdxWrite	:= iTotalIdxWrite + 1;

			IF tyParameter.tyAvl.a_tyUpstreamConfigurations[i].bUpstreamLaneId = TRUE THEN
				pa_tyXMLTable[iTotalIdxWrite].sTitle	:= 'AT';
				pa_tyXMLTable[iTotalIdxWrite].sValue	:= 'UpstreamLaneId';
				pa_tyXMLTable[iTotalIdxWrite].uiSize	:= LEN(pa_tyXMLTable[iTotalIdxWrite].sValue);

				iTotalIdxWrite	:= iTotalIdxWrite + 1;

				pa_tyXMLTable[iTotalIdxWrite].sTitle	:= 'AV';
				pa_tyXMLTable[iTotalIdxWrite].sValue	:= INT_TO_STRING(tyParameter.tyData.a_tyUpstreamConfigurations[i].iUpstreamLaneId);
				pa_tyXMLTable[iTotalIdxWrite].uiSize	:= LEN(pa_tyXMLTable[iTotalIdxWrite].sValue);

				iTotalIdxWrite	:= iTotalIdxWrite + 1;
			END_IF

			IF tyParameter.tyAvl.a_tyUpstreamConfigurations[i].bUpstreamInterfaceId = TRUE THEN
				pa_tyXMLTable[iTotalIdxWrite].sTitle	:= 'AT';
				pa_tyXMLTable[iTotalIdxWrite].sValue	:= 'UpstreamInterfaceId';
				pa_tyXMLTable[iTotalIdxWrite].uiSize	:= LEN(pa_tyXMLTable[iTotalIdxWrite].sValue);

				iTotalIdxWrite	:= iTotalIdxWrite + 1;

				pa_tyXMLTable[iTotalIdxWrite].sTitle	:= 'AV';
				pa_tyXMLTable[iTotalIdxWrite].sValue	:= tyParameter.tyData.a_tyUpstreamConfigurations[i].sUpstreamInterfaceId;
				pa_tyXMLTable[iTotalIdxWrite].uiSize	:= LEN(pa_tyXMLTable[iTotalIdxWrite].sValue);

				iTotalIdxWrite	:= iTotalIdxWrite + 1;
			END_IF

			IF tyParameter.tyAvl.a_tyUpstreamConfigurations[i].bHostAddress = TRUE THEN
				pa_tyXMLTable[iTotalIdxWrite].sTitle	:= 'AT';
				pa_tyXMLTable[iTotalIdxWrite].sValue	:= 'HostAddress';
				pa_tyXMLTable[iTotalIdxWrite].uiSize	:= LEN(pa_tyXMLTable[iTotalIdxWrite].sValue);

				iTotalIdxWrite	:= iTotalIdxWrite + 1;

				pa_tyXMLTable[iTotalIdxWrite].sTitle	:= 'AV';
				pa_tyXMLTable[iTotalIdxWrite].sValue	:= tyParameter.tyData.a_tyUpstreamConfigurations[i].sHostAddress;
				pa_tyXMLTable[iTotalIdxWrite].uiSize	:= LEN(pa_tyXMLTable[iTotalIdxWrite].sValue);

				iTotalIdxWrite	:= iTotalIdxWrite + 1;
			END_IF

			IF tyParameter.tyAvl.a_tyUpstreamConfigurations[i].bPort = TRUE THEN
				pa_tyXMLTable[iTotalIdxWrite].sTitle	:= 'AT';
				pa_tyXMLTable[iTotalIdxWrite].sValue	:= 'Port';
				pa_tyXMLTable[iTotalIdxWrite].uiSize	:= LEN(pa_tyXMLTable[iTotalIdxWrite].sValue);

				iTotalIdxWrite	:= iTotalIdxWrite + 1;

				pa_tyXMLTable[iTotalIdxWrite].sTitle	:= 'AV';
				pa_tyXMLTable[iTotalIdxWrite].sValue	:= UINT_TO_STRING(tyParameter.tyData.a_tyUpstreamConfigurations[i].uiPort);
				pa_tyXMLTable[iTotalIdxWrite].uiSize	:= LEN(pa_tyXMLTable[iTotalIdxWrite].sValue);

				iTotalIdxWrite	:= iTotalIdxWrite + 1;
			END_IF

			pa_tyXMLTable[iTotalIdxWrite].sTitle	:= 'ES';
			pa_tyXMLTable[iTotalIdxWrite].sValue	:= '';
			pa_tyXMLTable[iTotalIdxWrite].uiSize	:= LEN(pa_tyXMLTable[iTotalIdxWrite].sValue);

			iTotalIdxWrite	:= iTotalIdxWrite + 1;

		END_FOR

		pa_tyXMLTable[iTotalIdxWrite].sTitle	:= 'ET';
		pa_tyXMLTable[iTotalIdxWrite].sValue	:= 'UpstreamConfigurations';
		pa_tyXMLTable[iTotalIdxWrite].uiSize	:= LEN(pa_tyXMLTable[iTotalIdxWrite].sValue);

		iTotalIdxWrite	:= iTotalIdxWrite + 1;

		pa_tyXMLTable[iTotalIdxWrite].sTitle	:= 'EN';
		pa_tyXMLTable[iTotalIdxWrite].sValue	:= '';
		pa_tyXMLTable[iTotalIdxWrite].uiSize	:= LEN(pa_tyXMLTable[iTotalIdxWrite].sValue);

		iTotalIdxWrite	:= iTotalIdxWrite + 1;

	END_IF

	IF tyParameter.tyAvl.iDownstreamConfigurations > 0 THEN

		pa_tyXMLTable[iTotalIdxWrite].sTitle	:= 'ST';
		pa_tyXMLTable[iTotalIdxWrite].sValue	:= 'DownstreamConfigurations';
		pa_tyXMLTable[iTotalIdxWrite].uiSize	:= LEN(pa_tyXMLTable[iTotalIdxWrite].sValue);

		iTotalIdxWrite	:= iTotalIdxWrite + 1;

		pa_tyXMLTable[iTotalIdxWrite].sTitle	:= 'EN';
		pa_tyXMLTable[iTotalIdxWrite].sValue	:= '';
		pa_tyXMLTable[iTotalIdxWrite].uiSize	:= LEN(pa_tyXMLTable[iTotalIdxWrite].sValue);

		iTotalIdxWrite	:= iTotalIdxWrite + 1;

		IF tyParameter.tyAvl.iDownstreamConfigurations < 4 THEN
			iConfiguration	:= tyParameter.tyAvl.iDownstreamConfigurations - 1;
		ELSE
			iConfiguration	:= 2;
		END_IF

		FOR i := 0 TO iConfiguration DO

			pa_tyXMLTable[iTotalIdxWrite].sTitle	:= 'ST';
			pa_tyXMLTable[iTotalIdxWrite].sValue	:= 'DownstreamConfiguration';
			pa_tyXMLTable[iTotalIdxWrite].uiSize	:= LEN(pa_tyXMLTable[iTotalIdxWrite].sValue);

			iTotalIdxWrite	:= iTotalIdxWrite + 1;

			IF tyParameter.tyAvl.a_tyDownstreamConfigurations[i].bDownstreamLaneId = TRUE THEN
				pa_tyXMLTable[iTotalIdxWrite].sTitle	:= 'AT';
				pa_tyXMLTable[iTotalIdxWrite].sValue	:= 'DownstreamLaneId';
				pa_tyXMLTable[iTotalIdxWrite].uiSize	:= LEN(pa_tyXMLTable[iTotalIdxWrite].sValue);

				iTotalIdxWrite	:= iTotalIdxWrite + 1;

				pa_tyXMLTable[iTotalIdxWrite].sTitle	:= 'AV';
				pa_tyXMLTable[iTotalIdxWrite].sValue	:= INT_TO_STRING(tyParameter.tyData.a_tyDownstreamConfigurations[i].iDownstreamLaneId);
				pa_tyXMLTable[iTotalIdxWrite].uiSize	:= LEN(pa_tyXMLTable[iTotalIdxWrite].sValue);

				iTotalIdxWrite	:= iTotalIdxWrite + 1;
			END_IF

			IF tyParameter.tyAvl.a_tyDownstreamConfigurations[i].bDownstreamInterfaceId = TRUE THEN
				pa_tyXMLTable[iTotalIdxWrite].sTitle	:= 'AT';
				pa_tyXMLTable[iTotalIdxWrite].sValue	:= 'DownstreamInterfaceId';
				pa_tyXMLTable[iTotalIdxWrite].uiSize	:= LEN(pa_tyXMLTable[iTotalIdxWrite].sValue);

				iTotalIdxWrite	:= iTotalIdxWrite + 1;

				pa_tyXMLTable[iTotalIdxWrite].sTitle	:= 'AV';
				pa_tyXMLTable[iTotalIdxWrite].sValue	:= tyParameter.tyData.a_tyDownstreamConfigurations[i].sDownstreamInterfaceId;
				pa_tyXMLTable[iTotalIdxWrite].uiSize	:= LEN(pa_tyXMLTable[iTotalIdxWrite].sValue);

				iTotalIdxWrite	:= iTotalIdxWrite + 1;
			END_IF

			IF tyParameter.tyAvl.a_tyDownstreamConfigurations[i].bClientAddress = TRUE THEN
				pa_tyXMLTable[iTotalIdxWrite].sTitle	:= 'AT';
				pa_tyXMLTable[iTotalIdxWrite].sValue	:= 'ClientAddress';
				pa_tyXMLTable[iTotalIdxWrite].uiSize	:= LEN(pa_tyXMLTable[iTotalIdxWrite].sValue);

				iTotalIdxWrite	:= iTotalIdxWrite + 1;

				pa_tyXMLTable[iTotalIdxWrite].sTitle	:= 'AV';
				pa_tyXMLTable[iTotalIdxWrite].sValue	:= tyParameter.tyData.a_tyDownstreamConfigurations[i].sClientAddress;
				pa_tyXMLTable[iTotalIdxWrite].uiSize	:= LEN(pa_tyXMLTable[iTotalIdxWrite].sValue);

				iTotalIdxWrite	:= iTotalIdxWrite + 1;
			END_IF

			IF tyParameter.tyAvl.a_tyDownstreamConfigurations[i].bPort = TRUE THEN
				pa_tyXMLTable[iTotalIdxWrite].sTitle	:= 'AT';
				pa_tyXMLTable[iTotalIdxWrite].sValue	:= 'Port';
				pa_tyXMLTable[iTotalIdxWrite].uiSize	:= LEN(pa_tyXMLTable[iTotalIdxWrite].sValue);

				iTotalIdxWrite	:= iTotalIdxWrite + 1;

				pa_tyXMLTable[iTotalIdxWrite].sTitle	:= 'AV';
				pa_tyXMLTable[iTotalIdxWrite].sValue	:= UINT_TO_STRING(tyParameter.tyData.a_tyDownstreamConfigurations[i].uiPort);
				pa_tyXMLTable[iTotalIdxWrite].uiSize	:= LEN(pa_tyXMLTable[iTotalIdxWrite].sValue);

				iTotalIdxWrite	:= iTotalIdxWrite + 1;
			END_IF

			pa_tyXMLTable[iTotalIdxWrite].sTitle	:= 'ES';
			pa_tyXMLTable[iTotalIdxWrite].sValue	:= '';
			pa_tyXMLTable[iTotalIdxWrite].uiSize	:= LEN(pa_tyXMLTable[iTotalIdxWrite].sValue);

			iTotalIdxWrite	:= iTotalIdxWrite + 1;

		END_FOR

		pa_tyXMLTable[iTotalIdxWrite].sTitle	:= 'ET';
		pa_tyXMLTable[iTotalIdxWrite].sValue	:= 'DownstreamConfigurations';
		pa_tyXMLTable[iTotalIdxWrite].uiSize	:= LEN(pa_tyXMLTable[iTotalIdxWrite].sValue);

		iTotalIdxWrite	:= iTotalIdxWrite + 1;

		pa_tyXMLTable[iTotalIdxWrite].sTitle	:= 'EN';
		pa_tyXMLTable[iTotalIdxWrite].sValue	:= '';
		pa_tyXMLTable[iTotalIdxWrite].uiSize	:= LEN(pa_tyXMLTable[iTotalIdxWrite].sValue);

		iTotalIdxWrite	:= iTotalIdxWrite + 1;

	END_IF

	pa_tyXMLTable[iTotalIdxWrite].sTitle	:= 'ET';
	pa_tyXMLTable[iTotalIdxWrite].sValue	:= 'SetConfiguration';
	pa_tyXMLTable[iTotalIdxWrite].uiSize	:= LEN(pa_tyXMLTable[iTotalIdxWrite].sValue);

	iTotalIdxWrite	:= iTotalIdxWrite + 1;

	pa_tyXMLTable[iTotalIdxWrite].sTitle	:= 'EN';
	pa_tyXMLTable[iTotalIdxWrite].sValue	:= '';
	pa_tyXMLTable[iTotalIdxWrite].uiSize	:= LEN(pa_tyXMLTable[iTotalIdxWrite].sValue);

	iTotalIdxWrite	:= iTotalIdxWrite + 1;

	pa_tyXMLTable[iTotalIdxWrite].sTitle	:= 'ET';
	pa_tyXMLTable[iTotalIdxWrite].sValue	:= 'Hermes';
	pa_tyXMLTable[iTotalIdxWrite].uiSize	:= LEN(pa_tyXMLTable[iTotalIdxWrite].sValue);

	iTotalIdxWrite	:= iTotalIdxWrite + 1;

	pa_tyXMLTable[iTotalIdxWrite].sTitle	:= 'EN';
	pa_tyXMLTable[iTotalIdxWrite].sValue	:= '';
	pa_tyXMLTable[iTotalIdxWrite].uiSize	:= LEN(pa_tyXMLTable[iTotalIdxWrite].sValue);

	iTotalIdxWrite	:= iTotalIdxWrite + 1;

	iTotalIdxWrite	:= fHermesFormSetConfiguration;

END_FUNCTION
```

#### fHermesFormGetConfiguration.st
```iecst
(* Hermes Form Get Configuration Table Data (Total Index Written In Table) *)
FUNCTION fHermesFormGetConfiguration

	memset(ADR(pa_tyXMLTable) , 0 , SIZEOF(pa_tyXMLTable));
	iTotalIdxWrite	:= 0;

	fHermesGetTimestamp(ADR(sTimestamp) , tyDTStructure);

	pa_tyXMLTable[iTotalIdxWrite].sTitle	:= 'ST';
	pa_tyXMLTable[iTotalIdxWrite].sValue	:= 'Hermes';
	pa_tyXMLTable[iTotalIdxWrite].uiSize	:= LEN(pa_tyXMLTable[iTotalIdxWrite].sValue);

	iTotalIdxWrite	:= iTotalIdxWrite + 1;

	pa_tyXMLTable[iTotalIdxWrite].sTitle	:= 'AT';
	pa_tyXMLTable[iTotalIdxWrite].sValue	:= 'Timestamp';
	pa_tyXMLTable[iTotalIdxWrite].uiSize	:= LEN(pa_tyXMLTable[iTotalIdxWrite].sValue);

	iTotalIdxWrite	:= iTotalIdxWrite + 1;

	pa_tyXMLTable[iTotalIdxWrite].sTitle	:= 'AV';
	pa_tyXMLTable[iTotalIdxWrite].sValue	:= sTimestamp;
	pa_tyXMLTable[iTotalIdxWrite].uiSize	:= LEN(pa_tyXMLTable[iTotalIdxWrite].sValue);

	iTotalIdxWrite	:= iTotalIdxWrite + 1;

	pa_tyXMLTable[iTotalIdxWrite].sTitle	:= 'EN';
	pa_tyXMLTable[iTotalIdxWrite].sValue	:= '';
	pa_tyXMLTable[iTotalIdxWrite].uiSize	:= LEN(pa_tyXMLTable[iTotalIdxWrite].sValue);

	iTotalIdxWrite	:= iTotalIdxWrite + 1;

	pa_tyXMLTable[iTotalIdxWrite].sTitle	:= 'ST';
	pa_tyXMLTable[iTotalIdxWrite].sValue	:= 'GetConfiguration';
	pa_tyXMLTable[iTotalIdxWrite].uiSize	:= LEN(pa_tyXMLTable[iTotalIdxWrite].sValue);

	iTotalIdxWrite	:= iTotalIdxWrite + 1;

	pa_tyXMLTable[iTotalIdxWrite].sTitle	:= 'ES';
	pa_tyXMLTable[iTotalIdxWrite].sValue	:= '';
	pa_tyXMLTable[iTotalIdxWrite].uiSize	:= LEN(pa_tyXMLTable[iTotalIdxWrite].sValue);

	iTotalIdxWrite	:= iTotalIdxWrite + 1;

	pa_tyXMLTable[iTotalIdxWrite].sTitle	:= 'ET';
	pa_tyXMLTable[iTotalIdxWrite].sValue	:= 'Hermes';
	pa_tyXMLTable[iTotalIdxWrite].uiSize	:= LEN(pa_tyXMLTable[iTotalIdxWrite].sValue);

	iTotalIdxWrite	:= iTotalIdxWrite + 1;

	pa_tyXMLTable[iTotalIdxWrite].sTitle	:= 'EN';
	pa_tyXMLTable[iTotalIdxWrite].sValue	:= '';
	pa_tyXMLTable[iTotalIdxWrite].uiSize	:= LEN(pa_tyXMLTable[iTotalIdxWrite].sValue);

	iTotalIdxWrite	:= iTotalIdxWrite + 1;

	iTotalIdxWrite	:= fHermesFormGetConfiguration;

END_FUNCTION
```

#### fHermesFormCurrentConfiguration.st
```iecst
(* Hermes Form Current Configuration Table Data (Total Index Written In Table) *)
FUNCTION fHermesFormCurrentConfiguration

	memset(ADR(pa_tyXMLTable) , 0 , SIZEOF(pa_tyXMLTable));
	iTotalIdxWrite	:= 0;

	fHermesGetTimestamp(ADR(sTimestamp) , tyDTStructure);

	pa_tyXMLTable[iTotalIdxWrite].sTitle	:= 'ST';
	pa_tyXMLTable[iTotalIdxWrite].sValue	:= 'Hermes';
	pa_tyXMLTable[iTotalIdxWrite].uiSize	:= LEN(pa_tyXMLTable[iTotalIdxWrite].sValue);

	iTotalIdxWrite	:= iTotalIdxWrite + 1;

	pa_tyXMLTable[iTotalIdxWrite].sTitle	:= 'AT';
	pa_tyXMLTable[iTotalIdxWrite].sValue	:= 'Timestamp';
	pa_tyXMLTable[iTotalIdxWrite].uiSize	:= LEN(pa_tyXMLTable[iTotalIdxWrite].sValue);

	iTotalIdxWrite	:= iTotalIdxWrite + 1;

	pa_tyXMLTable[iTotalIdxWrite].sTitle	:= 'AV';
	pa_tyXMLTable[iTotalIdxWrite].sValue	:= sTimestamp;
	pa_tyXMLTable[iTotalIdxWrite].uiSize	:= LEN(pa_tyXMLTable[iTotalIdxWrite].sValue);

	iTotalIdxWrite	:= iTotalIdxWrite + 1;

	pa_tyXMLTable[iTotalIdxWrite].sTitle	:= 'EN';
	pa_tyXMLTable[iTotalIdxWrite].sValue	:= '';
	pa_tyXMLTable[iTotalIdxWrite].uiSize	:= LEN(pa_tyXMLTable[iTotalIdxWrite].sValue);

	iTotalIdxWrite	:= iTotalIdxWrite + 1;

	pa_tyXMLTable[iTotalIdxWrite].sTitle	:= 'ST';
	pa_tyXMLTable[iTotalIdxWrite].sValue	:= 'CurrentConfiguration';
	pa_tyXMLTable[iTotalIdxWrite].uiSize	:= LEN(pa_tyXMLTable[iTotalIdxWrite].sValue);

	iTotalIdxWrite	:= iTotalIdxWrite + 1;

	IF tyParameter.tyAvl.bMachineId = TRUE THEN
		pa_tyXMLTable[iTotalIdxWrite].sTitle	:= 'AT';
		pa_tyXMLTable[iTotalIdxWrite].sValue	:= 'MachineId';
		pa_tyXMLTable[iTotalIdxWrite].uiSize	:= LEN(pa_tyXMLTable[iTotalIdxWrite].sValue);

		iTotalIdxWrite	:= iTotalIdxWrite + 1;

		pa_tyXMLTable[iTotalIdxWrite].sTitle	:= 'AV';
		pa_tyXMLTable[iTotalIdxWrite].sValue	:= tyParameter.tyData.sMachineId;
		pa_tyXMLTable[iTotalIdxWrite].uiSize	:= LEN(pa_tyXMLTable[iTotalIdxWrite].sValue);

		iTotalIdxWrite	:= iTotalIdxWrite + 1;
	END_IF

	IF tyParameter.tyAvl.bMachineId = TRUE THEN
		pa_tyXMLTable[iTotalIdxWrite].sTitle	:= 'AT';
		pa_tyXMLTable[iTotalIdxWrite].sValue	:= 'SupervisorySystemPort';
		pa_tyXMLTable[iTotalIdxWrite].uiSize	:= LEN(pa_tyXMLTable[iTotalIdxWrite].sValue);

		iTotalIdxWrite	:= iTotalIdxWrite + 1;

		pa_tyXMLTable[iTotalIdxWrite].sTitle	:= 'AV';
		pa_tyXMLTable[iTotalIdxWrite].sValue	:= UINT_TO_STRING(tyParameter.tyData.uiSupervisorySystemPort);
		pa_tyXMLTable[iTotalIdxWrite].uiSize	:= LEN(pa_tyXMLTable[iTotalIdxWrite].sValue);

		iTotalIdxWrite	:= iTotalIdxWrite + 1;
	END_IF

	pa_tyXMLTable[iTotalIdxWrite].sTitle	:= 'EN';
	pa_tyXMLTable[iTotalIdxWrite].sValue	:= '';
	pa_tyXMLTable[iTotalIdxWrite].uiSize	:= LEN(pa_tyXMLTable[iTotalIdxWrite].sValue);

	iTotalIdxWrite	:= iTotalIdxWrite + 1;

	IF tyParameter.tyAvl.iUpstreamConfigurations > 0 THEN

		pa_tyXMLTable[iTotalIdxWrite].sTitle	:= 'ST';
		pa_tyXMLTable[iTotalIdxWrite].sValue	:= 'UpstreamConfigurations';
		pa_tyXMLTable[iTotalIdxWrite].uiSize	:= LEN(pa_tyXMLTable[iTotalIdxWrite].sValue);

		iTotalIdxWrite	:= iTotalIdxWrite + 1;

		pa_tyXMLTable[iTotalIdxWrite].sTitle	:= 'EN';
		pa_tyXMLTable[iTotalIdxWrite].sValue	:= '';
		pa_tyXMLTable[iTotalIdxWrite].uiSize	:= LEN(pa_tyXMLTable[iTotalIdxWrite].sValue);

		iTotalIdxWrite	:= iTotalIdxWrite + 1;

		IF tyParameter.tyAvl.iUpstreamConfigurations < 5 THEN
			iConfiguration	:= tyParameter.tyAvl.iUpstreamConfigurations - 1;
		ELSE
			iConfiguration	:= 4;
		END_IF

		FOR i := 0 TO iConfiguration DO

			pa_tyXMLTable[iTotalIdxWrite].sTitle	:= 'ST';
			pa_tyXMLTable[iTotalIdxWrite].sValue	:= 'UpstreamConfiguration';
			pa_tyXMLTable[iTotalIdxWrite].uiSize	:= LEN(pa_tyXMLTable[iTotalIdxWrite].sValue);

			iTotalIdxWrite	:= iTotalIdxWrite + 1;

			IF tyParameter.tyAvl.a_tyUpstreamConfigurations[i].bUpstreamLaneId = TRUE THEN
				pa_tyXMLTable[iTotalIdxWrite].sTitle	:= 'AT';
				pa_tyXMLTable[iTotalIdxWrite].sValue	:= 'UpstreamLaneId';
				pa_tyXMLTable[iTotalIdxWrite].uiSize	:= LEN(pa_tyXMLTable[iTotalIdxWrite].sValue);

				iTotalIdxWrite	:= iTotalIdxWrite + 1;

				pa_tyXMLTable[iTotalIdxWrite].sTitle	:= 'AV';
				pa_tyXMLTable[iTotalIdxWrite].sValue	:= INT_TO_STRING(tyParameter.tyData.a_tyUpstreamConfigurations[i].iUpstreamLaneId);
				pa_tyXMLTable[iTotalIdxWrite].uiSize	:= LEN(pa_tyXMLTable[iTotalIdxWrite].sValue);

				iTotalIdxWrite	:= iTotalIdxWrite + 1;
			END_IF

			IF tyParameter.tyAvl.a_tyUpstreamConfigurations[i].bUpstreamInterfaceId = TRUE THEN
				pa_tyXMLTable[iTotalIdxWrite].sTitle	:= 'AT';
				pa_tyXMLTable[iTotalIdxWrite].sValue	:= 'UpstreamInterfaceId';
				pa_tyXMLTable[iTotalIdxWrite].uiSize	:= LEN(pa_tyXMLTable[iTotalIdxWrite].sValue);

				iTotalIdxWrite	:= iTotalIdxWrite + 1;

				pa_tyXMLTable[iTotalIdxWrite].sTitle	:= 'AV';
				pa_tyXMLTable[iTotalIdxWrite].sValue	:= tyParameter.tyData.a_tyUpstreamConfigurations[i].sUpstreamInterfaceId;
				pa_tyXMLTable[iTotalIdxWrite].uiSize	:= LEN(pa_tyXMLTable[iTotalIdxWrite].sValue);

				iTotalIdxWrite	:= iTotalIdxWrite + 1;
			END_IF

			IF tyParameter.tyAvl.a_tyUpstreamConfigurations[i].bHostAddress = TRUE THEN
				pa_tyXMLTable[iTotalIdxWrite].sTitle	:= 'AT';
				pa_tyXMLTable[iTotalIdxWrite].sValue	:= 'HostAddress';
				pa_tyXMLTable[iTotalIdxWrite].uiSize	:= LEN(pa_tyXMLTable[iTotalIdxWrite].sValue);

				iTotalIdxWrite	:= iTotalIdxWrite + 1;

				pa_tyXMLTable[iTotalIdxWrite].sTitle	:= 'AV';
				pa_tyXMLTable[iTotalIdxWrite].sValue	:= tyParameter.tyData.a_tyUpstreamConfigurations[i].sHostAddress;
				pa_tyXMLTable[iTotalIdxWrite].uiSize	:= LEN(pa_tyXMLTable[iTotalIdxWrite].sValue);

				iTotalIdxWrite	:= iTotalIdxWrite + 1;
			END_IF

			IF tyParameter.tyAvl.a_tyUpstreamConfigurations[i].bPort = TRUE THEN
				pa_tyXMLTable[iTotalIdxWrite].sTitle	:= 'AT';
				pa_tyXMLTable[iTotalIdxWrite].sValue	:= 'Port';
				pa_tyXMLTable[iTotalIdxWrite].uiSize	:= LEN(pa_tyXMLTable[iTotalIdxWrite].sValue);

				iTotalIdxWrite	:= iTotalIdxWrite + 1;

				pa_tyXMLTable[iTotalIdxWrite].sTitle	:= 'AV';
				pa_tyXMLTable[iTotalIdxWrite].sValue	:= UINT_TO_STRING(tyParameter.tyData.a_tyUpstreamConfigurations[i].uiPort);
				pa_tyXMLTable[iTotalIdxWrite].uiSize	:= LEN(pa_tyXMLTable[iTotalIdxWrite].sValue);

				iTotalIdxWrite	:= iTotalIdxWrite + 1;
			END_IF

			pa_tyXMLTable[iTotalIdxWrite].sTitle	:= 'ES';
			pa_tyXMLTable[iTotalIdxWrite].sValue	:= '';
			pa_tyXMLTable[iTotalIdxWrite].uiSize	:= LEN(pa_tyXMLTable[iTotalIdxWrite].sValue);

			iTotalIdxWrite	:= iTotalIdxWrite + 1;

		END_FOR

		pa_tyXMLTable[iTotalIdxWrite].sTitle	:= 'ET';
		pa_tyXMLTable[iTotalIdxWrite].sValue	:= 'UpstreamConfigurations';
		pa_tyXMLTable[iTotalIdxWrite].uiSize	:= LEN(pa_tyXMLTable[iTotalIdxWrite].sValue);

		iTotalIdxWrite	:= iTotalIdxWrite + 1;

		pa_tyXMLTable[iTotalIdxWrite].sTitle	:= 'EN';
		pa_tyXMLTable[iTotalIdxWrite].sValue	:= '';
		pa_tyXMLTable[iTotalIdxWrite].uiSize	:= LEN(pa_tyXMLTable[iTotalIdxWrite].sValue);

		iTotalIdxWrite	:= iTotalIdxWrite + 1;

	END_IF

	IF tyParameter.tyAvl.iDownstreamConfigurations > 0 THEN

		pa_tyXMLTable[iTotalIdxWrite].sTitle	:= 'ST';
		pa_tyXMLTable[iTotalIdxWrite].sValue	:= 'DownstreamConfigurations';
		pa_tyXMLTable[iTotalIdxWrite].uiSize	:= LEN(pa_tyXMLTable[iTotalIdxWrite].sValue);

		iTotalIdxWrite	:= iTotalIdxWrite + 1;

		pa_tyXMLTable[iTotalIdxWrite].sTitle	:= 'EN';
		pa_tyXMLTable[iTotalIdxWrite].sValue	:= '';
		pa_tyXMLTable[iTotalIdxWrite].uiSize	:= LEN(pa_tyXMLTable[iTotalIdxWrite].sValue);

		iTotalIdxWrite	:= iTotalIdxWrite + 1;

		IF tyParameter.tyAvl.iDownstreamConfigurations < 5 THEN
			iConfiguration1	:= tyParameter.tyAvl.iDownstreamConfigurations - 1;
		ELSE
			iConfiguration1	:= 4;
		END_IF

		FOR i := 0 TO iConfiguration1 DO

			pa_tyXMLTable[iTotalIdxWrite].sTitle	:= 'ST';
			pa_tyXMLTable[iTotalIdxWrite].sValue	:= 'DownstreamConfiguration';
			pa_tyXMLTable[iTotalIdxWrite].uiSize	:= LEN(pa_tyXMLTable[iTotalIdxWrite].sValue);

			iTotalIdxWrite	:= iTotalIdxWrite + 1;

			IF tyParameter.tyAvl.a_tyDownstreamConfigurations[i].bDownstreamLaneId = TRUE THEN
				pa_tyXMLTable[iTotalIdxWrite].sTitle	:= 'AT';
				pa_tyXMLTable[iTotalIdxWrite].sValue	:= 'DownstreamLaneId';
				pa_tyXMLTable[iTotalIdxWrite].uiSize	:= LEN(pa_tyXMLTable[iTotalIdxWrite].sValue);

				iTotalIdxWrite	:= iTotalIdxWrite + 1;

				pa_tyXMLTable[iTotalIdxWrite].sTitle	:= 'AV';
				pa_tyXMLTable[iTotalIdxWrite].sValue	:= INT_TO_STRING(tyParameter.tyData.a_tyDownstreamConfigurations[i].iDownstreamLaneId);
				pa_tyXMLTable[iTotalIdxWrite].uiSize	:= LEN(pa_tyXMLTable[iTotalIdxWrite].sValue);

				iTotalIdxWrite	:= iTotalIdxWrite + 1;
			END_IF

			IF tyParameter.tyAvl.a_tyDownstreamConfigurations[i].bDownstreamInterfaceId = TRUE THEN
				pa_tyXMLTable[iTotalIdxWrite].sTitle	:= 'AT';
				pa_tyXMLTable[iTotalIdxWrite].sValue	:= 'DownstreamInterfaceId';
				pa_tyXMLTable[iTotalIdxWrite].uiSize	:= LEN(pa_tyXMLTable[iTotalIdxWrite].sValue);

				iTotalIdxWrite	:= iTotalIdxWrite + 1;

				pa_tyXMLTable[iTotalIdxWrite].sTitle	:= 'AV';
				pa_tyXMLTable[iTotalIdxWrite].sValue	:= tyParameter.tyData.a_tyDownstreamConfigurations[i].sDownstreamInterfaceId;
				pa_tyXMLTable[iTotalIdxWrite].uiSize	:= LEN(pa_tyXMLTable[iTotalIdxWrite].sValue);

				iTotalIdxWrite	:= iTotalIdxWrite + 1;
			END_IF

			IF tyParameter.tyAvl.a_tyDownstreamConfigurations[i].bClientAddress = TRUE THEN
				pa_tyXMLTable[iTotalIdxWrite].sTitle	:= 'AT';
				pa_tyXMLTable[iTotalIdxWrite].sValue	:= 'ClientAddress';
				pa_tyXMLTable[iTotalIdxWrite].uiSize	:= LEN(pa_tyXMLTable[iTotalIdxWrite].sValue);

				iTotalIdxWrite	:= iTotalIdxWrite + 1;

				pa_tyXMLTable[iTotalIdxWrite].sTitle	:= 'AV';
				pa_tyXMLTable[iTotalIdxWrite].sValue	:= tyParameter.tyData.a_tyDownstreamConfigurations[i].sClientAddress;
				pa_tyXMLTable[iTotalIdxWrite].uiSize	:= LEN(pa_tyXMLTable[iTotalIdxWrite].sValue);

				iTotalIdxWrite	:= iTotalIdxWrite + 1;
			END_IF

			IF tyParameter.tyAvl.a_tyDownstreamConfigurations[i].bPort = TRUE THEN
				pa_tyXMLTable[iTotalIdxWrite].sTitle	:= 'AT';
				pa_tyXMLTable[iTotalIdxWrite].sValue	:= 'Port';
				pa_tyXMLTable[iTotalIdxWrite].uiSize	:= LEN(pa_tyXMLTable[iTotalIdxWrite].sValue);

				iTotalIdxWrite	:= iTotalIdxWrite + 1;

				pa_tyXMLTable[iTotalIdxWrite].sTitle	:= 'AV';
				pa_tyXMLTable[iTotalIdxWrite].sValue	:= UINT_TO_STRING(tyParameter.tyData.a_tyDownstreamConfigurations[i].uiPort);
				pa_tyXMLTable[iTotalIdxWrite].uiSize	:= LEN(pa_tyXMLTable[iTotalIdxWrite].sValue);

				iTotalIdxWrite	:= iTotalIdxWrite + 1;
			END_IF

			pa_tyXMLTable[iTotalIdxWrite].sTitle	:= 'ES';
			pa_tyXMLTable[iTotalIdxWrite].sValue	:= '';
			pa_tyXMLTable[iTotalIdxWrite].uiSize	:= LEN(pa_tyXMLTable[iTotalIdxWrite].sValue);

			iTotalIdxWrite	:= iTotalIdxWrite + 1;

		END_FOR

		pa_tyXMLTable[iTotalIdxWrite].sTitle	:= 'ET';
		pa_tyXMLTable[iTotalIdxWrite].sValue	:= 'DownstreamConfigurations';
		pa_tyXMLTable[iTotalIdxWrite].uiSize	:= LEN(pa_tyXMLTable[iTotalIdxWrite].sValue);

		iTotalIdxWrite	:= iTotalIdxWrite + 1;

		pa_tyXMLTable[iTotalIdxWrite].sTitle	:= 'EN';
		pa_tyXMLTable[iTotalIdxWrite].sValue	:= '';
		pa_tyXMLTable[iTotalIdxWrite].uiSize	:= LEN(pa_tyXMLTable[iTotalIdxWrite].sValue);

		iTotalIdxWrite	:= iTotalIdxWrite + 1;

	END_IF

	pa_tyXMLTable[iTotalIdxWrite].sTitle	:= 'ET';
	pa_tyXMLTable[iTotalIdxWrite].sValue	:= 'CurrentConfiguration';
	pa_tyXMLTable[iTotalIdxWrite].uiSize	:= LEN(pa_tyXMLTable[iTotalIdxWrite].sValue);

	iTotalIdxWrite	:= iTotalIdxWrite + 1;

	pa_tyXMLTable[iTotalIdxWrite].sTitle	:= 'EN';
	pa_tyXMLTable[iTotalIdxWrite].sValue	:= '';
	pa_tyXMLTable[iTotalIdxWrite].uiSize	:= LEN(pa_tyXMLTable[iTotalIdxWrite].sValue);

	iTotalIdxWrite	:= iTotalIdxWrite + 1;

	pa_tyXMLTable[iTotalIdxWrite].sTitle	:= 'ET';
	pa_tyXMLTable[iTotalIdxWrite].sValue	:= 'Hermes';
	pa_tyXMLTable[iTotalIdxWrite].uiSize	:= LEN(pa_tyXMLTable[iTotalIdxWrite].sValue);

	iTotalIdxWrite	:= iTotalIdxWrite + 1;

	pa_tyXMLTable[iTotalIdxWrite].sTitle	:= 'EN';
	pa_tyXMLTable[iTotalIdxWrite].sValue	:= '';
	pa_tyXMLTable[iTotalIdxWrite].uiSize	:= LEN(pa_tyXMLTable[iTotalIdxWrite].sValue);

	iTotalIdxWrite	:= iTotalIdxWrite + 1;

	iTotalIdxWrite	:= fHermesFormCurrentConfiguration;

END_FUNCTION
```

#### fHermesFormBoardForecast.st
```iecst
(* Hermes Form Board Forecast Table Data (Total Index Written In Table) *)
FUNCTION fHermesFormBoardForecast

	memset(ADR(pa_tyXMLTable) , 0 , SIZEOF(pa_tyXMLTable));
	iTotalIdxWrite	:= 0;

	fHermesGetTimestamp(ADR(sTimestamp) , tyDTStructure);

	pa_tyXMLTable[iTotalIdxWrite].sTitle	:= 'ST';
	pa_tyXMLTable[iTotalIdxWrite].sValue	:= 'Hermes';
	pa_tyXMLTable[iTotalIdxWrite].uiSize	:= LEN(pa_tyXMLTable[iTotalIdxWrite].sValue);

	iTotalIdxWrite	:= iTotalIdxWrite + 1;

	pa_tyXMLTable[iTotalIdxWrite].sTitle	:= 'AT';
	pa_tyXMLTable[iTotalIdxWrite].sValue	:= 'Timestamp';
	pa_tyXMLTable[iTotalIdxWrite].uiSize	:= LEN(pa_tyXMLTable[iTotalIdxWrite].sValue);

	iTotalIdxWrite	:= iTotalIdxWrite + 1;

	pa_tyXMLTable[iTotalIdxWrite].sTitle	:= 'AV';
	pa_tyXMLTable[iTotalIdxWrite].sValue	:= sTimestamp;
	pa_tyXMLTable[iTotalIdxWrite].uiSize	:= LEN(pa_tyXMLTable[iTotalIdxWrite].sValue);

	iTotalIdxWrite	:= iTotalIdxWrite + 1;

	pa_tyXMLTable[iTotalIdxWrite].sTitle	:= 'EN';
	pa_tyXMLTable[iTotalIdxWrite].sValue	:= '';
	pa_tyXMLTable[iTotalIdxWrite].uiSize	:= LEN(pa_tyXMLTable[iTotalIdxWrite].sValue);

	iTotalIdxWrite	:= iTotalIdxWrite + 1;

	pa_tyXMLTable[iTotalIdxWrite].sTitle	:= 'ST';
	pa_tyXMLTable[iTotalIdxWrite].sValue	:= 'BoardForecast';
	pa_tyXMLTable[iTotalIdxWrite].uiSize	:= LEN(pa_tyXMLTable[iTotalIdxWrite].sValue);

	iTotalIdxWrite	:= iTotalIdxWrite + 1;

	IF tyParameter.tyAvl.bForecastId = TRUE THEN
		pa_tyXMLTable[iTotalIdxWrite].sTitle	:= 'AT';
		pa_tyXMLTable[iTotalIdxWrite].sValue	:= 'ForecastId';
		pa_tyXMLTable[iTotalIdxWrite].uiSize	:= LEN(pa_tyXMLTable[iTotalIdxWrite].sValue);

		iTotalIdxWrite	:= iTotalIdxWrite + 1;

		pa_tyXMLTable[iTotalIdxWrite].sTitle	:= 'AV';
		pa_tyXMLTable[iTotalIdxWrite].sValue	:= tyParameter.tyData.sForecastId;
		pa_tyXMLTable[iTotalIdxWrite].uiSize	:= LEN(pa_tyXMLTable[iTotalIdxWrite].sValue);

		iTotalIdxWrite	:= iTotalIdxWrite + 1;
	END_IF

	IF tyParameter.tyAvl.bTimeUntilAvailable = TRUE THEN
		pa_tyXMLTable[iTotalIdxWrite].sTitle	:= 'AT';
		pa_tyXMLTable[iTotalIdxWrite].sValue	:= 'TimeUntilAvailable';
		pa_tyXMLTable[iTotalIdxWrite].uiSize	:= LEN(pa_tyXMLTable[iTotalIdxWrite].sValue);

		iTotalIdxWrite	:= iTotalIdxWrite + 1;

		pa_tyXMLTable[iTotalIdxWrite].sTitle	:= 'AV';
		pa_tyXMLTable[iTotalIdxWrite].sValue	:= REAL_TO_STRING(tyParameter.tyData.rTimeUntilAvailable);
		pa_tyXMLTable[iTotalIdxWrite].uiSize	:= LEN(pa_tyXMLTable[iTotalIdxWrite].sValue);

		iTotalIdxWrite	:= iTotalIdxWrite + 1;
	END_IF

	IF tyParameter.tyAvl.bBoardId = TRUE THEN
		pa_tyXMLTable[iTotalIdxWrite].sTitle	:= 'AT';
		pa_tyXMLTable[iTotalIdxWrite].sValue	:= 'BoardId';
		pa_tyXMLTable[iTotalIdxWrite].uiSize	:= LEN(pa_tyXMLTable[iTotalIdxWrite].sValue);

		iTotalIdxWrite	:= iTotalIdxWrite + 1;

		pa_tyXMLTable[iTotalIdxWrite].sTitle	:= 'AV';
		pa_tyXMLTable[iTotalIdxWrite].sValue	:= tyParameter.tyData.sBoardId;
		pa_tyXMLTable[iTotalIdxWrite].uiSize	:= LEN(pa_tyXMLTable[iTotalIdxWrite].sValue);

		iTotalIdxWrite	:= iTotalIdxWrite + 1;
	END_IF

	IF tyParameter.tyAvl.bBoardIdCreatedBy = TRUE THEN
		pa_tyXMLTable[iTotalIdxWrite].sTitle	:= 'AT';
		pa_tyXMLTable[iTotalIdxWrite].sValue	:= 'BoardIdCreatedBy';
		pa_tyXMLTable[iTotalIdxWrite].uiSize	:= LEN(pa_tyXMLTable[iTotalIdxWrite].sValue);

		iTotalIdxWrite	:= iTotalIdxWrite + 1;

		pa_tyXMLTable[iTotalIdxWrite].sTitle	:= 'AV';
		pa_tyXMLTable[iTotalIdxWrite].sValue	:= tyParameter.tyData.sBoardIdCreatedBy;
		pa_tyXMLTable[iTotalIdxWrite].uiSize	:= LEN(pa_tyXMLTable[iTotalIdxWrite].sValue);

		iTotalIdxWrite	:= iTotalIdxWrite + 1;
	END_IF

	IF tyParameter.tyAvl.bFailedBoard = TRUE THEN
		pa_tyXMLTable[iTotalIdxWrite].sTitle	:= 'AT';
		pa_tyXMLTable[iTotalIdxWrite].sValue	:= 'FailedBoard';
		pa_tyXMLTable[iTotalIdxWrite].uiSize	:= LEN(pa_tyXMLTable[iTotalIdxWrite].sValue);

		iTotalIdxWrite	:= iTotalIdxWrite + 1;

		pa_tyXMLTable[iTotalIdxWrite].sTitle	:= 'AV';
		pa_tyXMLTable[iTotalIdxWrite].sValue	:= DINT_TO_STRING(UDINT_TO_DINT(tyParameter.tyData.eFailedBoard));
		pa_tyXMLTable[iTotalIdxWrite].uiSize	:= LEN(pa_tyXMLTable[iTotalIdxWrite].sValue);

		iTotalIdxWrite	:= iTotalIdxWrite + 1;
	END_IF

	IF tyParameter.tyAvl.bProductTypeId = TRUE THEN
		pa_tyXMLTable[iTotalIdxWrite].sTitle	:= 'AT';
		pa_tyXMLTable[iTotalIdxWrite].sValue	:= 'ProductTypeId';
		pa_tyXMLTable[iTotalIdxWrite].uiSize	:= LEN(pa_tyXMLTable[iTotalIdxWrite].sValue);

		iTotalIdxWrite	:= iTotalIdxWrite + 1;

		pa_tyXMLTable[iTotalIdxWrite].sTitle	:= 'AV';
		pa_tyXMLTable[iTotalIdxWrite].sValue	:= tyParameter.tyData.sProductTypeId;
		pa_tyXMLTable[iTotalIdxWrite].uiSize	:= LEN(pa_tyXMLTable[iTotalIdxWrite].sValue);

		iTotalIdxWrite	:= iTotalIdxWrite + 1;
	END_IF

	IF tyParameter.tyAvl.bFlippedBoard = TRUE THEN
		pa_tyXMLTable[iTotalIdxWrite].sTitle	:= 'AT';
		pa_tyXMLTable[iTotalIdxWrite].sValue	:= 'FlippedBoard';
		pa_tyXMLTable[iTotalIdxWrite].uiSize	:= LEN(pa_tyXMLTable[iTotalIdxWrite].sValue);

		iTotalIdxWrite	:= iTotalIdxWrite + 1;

		pa_tyXMLTable[iTotalIdxWrite].sTitle	:= 'AV';
		pa_tyXMLTable[iTotalIdxWrite].sValue	:= DINT_TO_STRING(UDINT_TO_DINT(tyParameter.tyData.eFlippedBoard));
		pa_tyXMLTable[iTotalIdxWrite].uiSize	:= LEN(pa_tyXMLTable[iTotalIdxWrite].sValue);

		iTotalIdxWrite	:= iTotalIdxWrite + 1;
	END_IF

	IF tyParameter.tyAvl.bTopBarcode = TRUE THEN
		pa_tyXMLTable[iTotalIdxWrite].sTitle	:= 'AT';
		pa_tyXMLTable[iTotalIdxWrite].sValue	:= 'TopBarcode';
		pa_tyXMLTable[iTotalIdxWrite].uiSize	:= LEN(pa_tyXMLTable[iTotalIdxWrite].sValue);

		iTotalIdxWrite	:= iTotalIdxWrite + 1;

		pa_tyXMLTable[iTotalIdxWrite].sTitle	:= 'AV';
		pa_tyXMLTable[iTotalIdxWrite].sValue	:= tyParameter.tyData.sTopBarcode;
		pa_tyXMLTable[iTotalIdxWrite].uiSize	:= LEN(pa_tyXMLTable[iTotalIdxWrite].sValue);

		iTotalIdxWrite	:= iTotalIdxWrite + 1;
	END_IF

	IF tyParameter.tyAvl.bBottomBarcode = TRUE THEN
		pa_tyXMLTable[iTotalIdxWrite].sTitle	:= 'AT';
		pa_tyXMLTable[iTotalIdxWrite].sValue	:= 'BottomBarcode';
		pa_tyXMLTable[iTotalIdxWrite].uiSize	:= LEN(pa_tyXMLTable[iTotalIdxWrite].sValue);

		iTotalIdxWrite	:= iTotalIdxWrite + 1;

		pa_tyXMLTable[iTotalIdxWrite].sTitle	:= 'AV';
		pa_tyXMLTable[iTotalIdxWrite].sValue	:= tyParameter.tyData.sBottomBarcode;
		pa_tyXMLTable[iTotalIdxWrite].uiSize	:= LEN(pa_tyXMLTable[iTotalIdxWrite].sValue);

		iTotalIdxWrite	:= iTotalIdxWrite + 1;
	END_IF

	IF tyParameter.tyAvl.bLength = TRUE THEN
		pa_tyXMLTable[iTotalIdxWrite].sTitle	:= 'AT';
		pa_tyXMLTable[iTotalIdxWrite].sValue	:= 'Length';
		pa_tyXMLTable[iTotalIdxWrite].uiSize	:= LEN(pa_tyXMLTable[iTotalIdxWrite].sValue);

		iTotalIdxWrite	:= iTotalIdxWrite + 1;

		pa_tyXMLTable[iTotalIdxWrite].sTitle	:= 'AV';
		pa_tyXMLTable[iTotalIdxWrite].sValue	:= REAL_TO_STRING(tyParameter.tyData.rLength);
		pa_tyXMLTable[iTotalIdxWrite].uiSize	:= LEN(pa_tyXMLTable[iTotalIdxWrite].sValue);

		iTotalIdxWrite	:= iTotalIdxWrite + 1;
	END_IF

	IF tyParameter.tyAvl.bWidth = TRUE THEN
		pa_tyXMLTable[iTotalIdxWrite].sTitle	:= 'AT';
		pa_tyXMLTable[iTotalIdxWrite].sValue	:= 'Width';
		pa_tyXMLTable[iTotalIdxWrite].uiSize	:= LEN(pa_tyXMLTable[iTotalIdxWrite].sValue);

		iTotalIdxWrite	:= iTotalIdxWrite + 1;

		pa_tyXMLTable[iTotalIdxWrite].sTitle	:= 'AV';
		pa_tyXMLTable[iTotalIdxWrite].sValue	:= REAL_TO_STRING(tyParameter.tyData.rWidth);
		pa_tyXMLTable[iTotalIdxWrite].uiSize	:= LEN(pa_tyXMLTable[iTotalIdxWrite].sValue);

		iTotalIdxWrite	:= iTotalIdxWrite + 1;
	END_IF

	IF tyParameter.tyAvl.bThickness = TRUE THEN
		pa_tyXMLTable[iTotalIdxWrite].sTitle	:= 'AT';
		pa_tyXMLTable[iTotalIdxWrite].sValue	:= 'Thickness';
		pa_tyXMLTable[iTotalIdxWrite].uiSize	:= LEN(pa_tyXMLTable[iTotalIdxWrite].sValue);

		iTotalIdxWrite	:= iTotalIdxWrite + 1;

		pa_tyXMLTable[iTotalIdxWrite].sTitle	:= 'AV';
		pa_tyXMLTable[iTotalIdxWrite].sValue	:= REAL_TO_STRING(tyParameter.tyData.rThickness);
		pa_tyXMLTable[iTotalIdxWrite].uiSize	:= LEN(pa_tyXMLTable[iTotalIdxWrite].sValue);

		iTotalIdxWrite	:= iTotalIdxWrite + 1;
	END_IF

	IF tyParameter.tyAvl.bConveyorSpeed = TRUE THEN
		pa_tyXMLTable[iTotalIdxWrite].sTitle	:= 'AT';
		pa_tyXMLTable[iTotalIdxWrite].sValue	:= 'ConveyorSpeed';
		pa_tyXMLTable[iTotalIdxWrite].uiSize	:= LEN(pa_tyXMLTable[iTotalIdxWrite].sValue);

		iTotalIdxWrite	:= iTotalIdxWrite + 1;

		pa_tyXMLTable[iTotalIdxWrite].sTitle	:= 'AV';
		pa_tyXMLTable[iTotalIdxWrite].sValue	:= REAL_TO_STRING(tyParameter.tyData.rConveyorSpeed);
		pa_tyXMLTable[iTotalIdxWrite].uiSize	:= LEN(pa_tyXMLTable[iTotalIdxWrite].sValue);

		iTotalIdxWrite	:= iTotalIdxWrite + 1;
	END_IF

	IF tyParameter.tyAvl.bTopClearanceHeight = TRUE THEN
		pa_tyXMLTable[iTotalIdxWrite].sTitle	:= 'AT';
		pa_tyXMLTable[iTotalIdxWrite].sValue	:= 'TopClearanceHeight';
		pa_tyXMLTable[iTotalIdxWrite].uiSize	:= LEN(pa_tyXMLTable[iTotalIdxWrite].sValue);

		iTotalIdxWrite	:= iTotalIdxWrite + 1;

		pa_tyXMLTable[iTotalIdxWrite].sTitle	:= 'AV';
		pa_tyXMLTable[iTotalIdxWrite].sValue	:= REAL_TO_STRING(tyParameter.tyData.rTopClearanceHeight);
		pa_tyXMLTable[iTotalIdxWrite].uiSize	:= LEN(pa_tyXMLTable[iTotalIdxWrite].sValue);

		iTotalIdxWrite	:= iTotalIdxWrite + 1;
	END_IF

	IF tyParameter.tyAvl.bBottomClearanceHeight = TRUE THEN
		pa_tyXMLTable[iTotalIdxWrite].sTitle	:= 'AT';
		pa_tyXMLTable[iTotalIdxWrite].sValue	:= 'BottomClearanceHeight';
		pa_tyXMLTable[iTotalIdxWrite].uiSize	:= LEN(pa_tyXMLTable[iTotalIdxWrite].sValue);

		iTotalIdxWrite	:= iTotalIdxWrite + 1;

		pa_tyXMLTable[iTotalIdxWrite].sTitle	:= 'AV';
		pa_tyXMLTable[iTotalIdxWrite].sValue	:= REAL_TO_STRING(tyParameter.tyData.rBottomClearanceHeight);
		pa_tyXMLTable[iTotalIdxWrite].uiSize	:= LEN(pa_tyXMLTable[iTotalIdxWrite].sValue);

		iTotalIdxWrite	:= iTotalIdxWrite + 1;
	END_IF

	IF tyParameter.tyAvl.bWeight = TRUE THEN
		pa_tyXMLTable[iTotalIdxWrite].sTitle	:= 'AT';
		pa_tyXMLTable[iTotalIdxWrite].sValue	:= 'Weight';
		pa_tyXMLTable[iTotalIdxWrite].uiSize	:= LEN(pa_tyXMLTable[iTotalIdxWrite].sValue);

		iTotalIdxWrite	:= iTotalIdxWrite + 1;

		pa_tyXMLTable[iTotalIdxWrite].sTitle	:= 'AV';
		pa_tyXMLTable[iTotalIdxWrite].sValue	:= REAL_TO_STRING(tyParameter.tyData.rWeight);
		pa_tyXMLTable[iTotalIdxWrite].uiSize	:= LEN(pa_tyXMLTable[iTotalIdxWrite].sValue);

		iTotalIdxWrite	:= iTotalIdxWrite + 1;
	END_IF

	IF tyParameter.tyAvl.bWorkOrderId = TRUE THEN
		pa_tyXMLTable[iTotalIdxWrite].sTitle	:= 'AT';
		pa_tyXMLTable[iTotalIdxWrite].sValue	:= 'WorkOrderId';
		pa_tyXMLTable[iTotalIdxWrite].uiSize	:= LEN(pa_tyXMLTable[iTotalIdxWrite].sValue);

		iTotalIdxWrite	:= iTotalIdxWrite + 1;

		pa_tyXMLTable[iTotalIdxWrite].sTitle	:= 'AV';
		pa_tyXMLTable[iTotalIdxWrite].sValue	:= tyParameter.tyData.sWorkOrderId;
		pa_tyXMLTable[iTotalIdxWrite].uiSize	:= LEN(pa_tyXMLTable[iTotalIdxWrite].sValue);

		iTotalIdxWrite	:= iTotalIdxWrite + 1;
	END_IF

	IF tyParameter.tyAvl.bBatchId = TRUE THEN
		pa_tyXMLTable[iTotalIdxWrite].sTitle	:= 'AT';
		pa_tyXMLTable[iTotalIdxWrite].sValue	:= 'BatchId';
		pa_tyXMLTable[iTotalIdxWrite].uiSize	:= LEN(pa_tyXMLTable[iTotalIdxWrite].sValue);

		iTotalIdxWrite	:= iTotalIdxWrite + 1;

		pa_tyXMLTable[iTotalIdxWrite].sTitle	:= 'AV';
		pa_tyXMLTable[iTotalIdxWrite].sValue	:= tyParameter.tyData.sBatchId;
		pa_tyXMLTable[iTotalIdxWrite].uiSize	:= LEN(pa_tyXMLTable[iTotalIdxWrite].sValue);

		iTotalIdxWrite	:= iTotalIdxWrite + 1;
	END_IF

	pa_tyXMLTable[iTotalIdxWrite].sTitle	:= 'ES';
	pa_tyXMLTable[iTotalIdxWrite].sValue	:= '';
	pa_tyXMLTable[iTotalIdxWrite].uiSize	:= LEN(pa_tyXMLTable[iTotalIdxWrite].sValue);

	iTotalIdxWrite	:= iTotalIdxWrite + 1;

	pa_tyXMLTable[iTotalIdxWrite].sTitle	:= 'ET';
	pa_tyXMLTable[iTotalIdxWrite].sValue	:= 'Hermes';
	pa_tyXMLTable[iTotalIdxWrite].uiSize	:= LEN(pa_tyXMLTable[iTotalIdxWrite].sValue);

	iTotalIdxWrite	:= iTotalIdxWrite + 1;

	pa_tyXMLTable[iTotalIdxWrite].sTitle	:= 'EN';
	pa_tyXMLTable[iTotalIdxWrite].sValue	:= '';
	pa_tyXMLTable[iTotalIdxWrite].uiSize	:= LEN(pa_tyXMLTable[iTotalIdxWrite].sValue);

	iTotalIdxWrite	:= iTotalIdxWrite + 1;

	iTotalIdxWrite	:= fHermesFormBoardForecast;

END_FUNCTION
```

#### fHermesFormQueryBoardInfo.st
```iecst
(* Hermes Form Query Board Info Table Data (Total Index Written In Table) *)
FUNCTION fHermesFormQueryBoardInfo

	memset(ADR(pa_tyXMLTable) , 0 , SIZEOF(pa_tyXMLTable));
	iTotalIdxWrite	:= 0;

	fHermesGetTimestamp(ADR(sTimestamp) , tyDTStructure);

	pa_tyXMLTable[iTotalIdxWrite].sTitle	:= 'ST';
	pa_tyXMLTable[iTotalIdxWrite].sValue	:= 'Hermes';
	pa_tyXMLTable[iTotalIdxWrite].uiSize	:= LEN(pa_tyXMLTable[iTotalIdxWrite].sValue);

	iTotalIdxWrite	:= iTotalIdxWrite + 1;

	pa_tyXMLTable[iTotalIdxWrite].sTitle	:= 'AT';
	pa_tyXMLTable[iTotalIdxWrite].sValue	:= 'Timestamp';
	pa_tyXMLTable[iTotalIdxWrite].uiSize	:= LEN(pa_tyXMLTable[iTotalIdxWrite].sValue);

	iTotalIdxWrite	:= iTotalIdxWrite + 1;

	pa_tyXMLTable[iTotalIdxWrite].sTitle	:= 'AV';
	pa_tyXMLTable[iTotalIdxWrite].sValue	:= sTimestamp;
	pa_tyXMLTable[iTotalIdxWrite].uiSize	:= LEN(pa_tyXMLTable[iTotalIdxWrite].sValue);

	iTotalIdxWrite	:= iTotalIdxWrite + 1;

	pa_tyXMLTable[iTotalIdxWrite].sTitle	:= 'EN';
	pa_tyXMLTable[iTotalIdxWrite].sValue	:= '';
	pa_tyXMLTable[iTotalIdxWrite].uiSize	:= LEN(pa_tyXMLTable[iTotalIdxWrite].sValue);

	iTotalIdxWrite	:= iTotalIdxWrite + 1;

	pa_tyXMLTable[iTotalIdxWrite].sTitle	:= 'ST';
	pa_tyXMLTable[iTotalIdxWrite].sValue	:= 'QueryBoardInfo';
	pa_tyXMLTable[iTotalIdxWrite].uiSize	:= LEN(pa_tyXMLTable[iTotalIdxWrite].sValue);

	iTotalIdxWrite	:= iTotalIdxWrite + 1;

	IF tyParameter.tyAvl.bTopBarcode = TRUE THEN
		pa_tyXMLTable[iTotalIdxWrite].sTitle	:= 'AT';
		pa_tyXMLTable[iTotalIdxWrite].sValue	:= 'TopBarcode';
		pa_tyXMLTable[iTotalIdxWrite].uiSize	:= LEN(pa_tyXMLTable[iTotalIdxWrite].sValue);

		iTotalIdxWrite	:= iTotalIdxWrite + 1;

		pa_tyXMLTable[iTotalIdxWrite].sTitle	:= 'AV';
		pa_tyXMLTable[iTotalIdxWrite].sValue	:= tyParameter.tyData.sTopBarcode;
		pa_tyXMLTable[iTotalIdxWrite].uiSize	:= LEN(pa_tyXMLTable[iTotalIdxWrite].sValue);

		iTotalIdxWrite	:= iTotalIdxWrite + 1;
	END_IF

	IF tyParameter.tyAvl.bBottomBarcode = TRUE THEN
		pa_tyXMLTable[iTotalIdxWrite].sTitle	:= 'AT';
		pa_tyXMLTable[iTotalIdxWrite].sValue	:= 'BottomBarcode';
		pa_tyXMLTable[iTotalIdxWrite].uiSize	:= LEN(pa_tyXMLTable[iTotalIdxWrite].sValue);

		iTotalIdxWrite	:= iTotalIdxWrite + 1;

		pa_tyXMLTable[iTotalIdxWrite].sTitle	:= 'AV';
		pa_tyXMLTable[iTotalIdxWrite].sValue	:= tyParameter.tyData.sBottomBarcode;
		pa_tyXMLTable[iTotalIdxWrite].uiSize	:= LEN(pa_tyXMLTable[iTotalIdxWrite].sValue);

		iTotalIdxWrite	:= iTotalIdxWrite + 1;
	END_IF

	pa_tyXMLTable[iTotalIdxWrite].sTitle	:= 'ES';
	pa_tyXMLTable[iTotalIdxWrite].sValue	:= '';
	pa_tyXMLTable[iTotalIdxWrite].uiSize	:= LEN(pa_tyXMLTable[iTotalIdxWrite].sValue);

	iTotalIdxWrite	:= iTotalIdxWrite + 1;

	pa_tyXMLTable[iTotalIdxWrite].sTitle	:= 'ET';
	pa_tyXMLTable[iTotalIdxWrite].sValue	:= 'Hermes';
	pa_tyXMLTable[iTotalIdxWrite].uiSize	:= LEN(pa_tyXMLTable[iTotalIdxWrite].sValue);

	iTotalIdxWrite	:= iTotalIdxWrite + 1;

	pa_tyXMLTable[iTotalIdxWrite].sTitle	:= 'EN';
	pa_tyXMLTable[iTotalIdxWrite].sValue	:= '';
	pa_tyXMLTable[iTotalIdxWrite].uiSize	:= LEN(pa_tyXMLTable[iTotalIdxWrite].sValue);

	iTotalIdxWrite	:= iTotalIdxWrite + 1;

	iTotalIdxWrite	:= fHermesFormQueryBoardInfo;

END_FUNCTION
```

#### fHermesFormSendBoardInfo.st
```iecst
(* Hermes Form Send Board Info Table Data (Total Index Written In Table) *)
FUNCTION fHermesFormSendBoardInfo

	memset(ADR(pa_tyXMLTable) , 0 , SIZEOF(pa_tyXMLTable));
	iTotalIdxWrite	:= 0;

	fHermesGetTimestamp(ADR(sTimestamp) , tyDTStructure);

	pa_tyXMLTable[iTotalIdxWrite].sTitle	:= 'ST';
	pa_tyXMLTable[iTotalIdxWrite].sValue	:= 'Hermes';
	pa_tyXMLTable[iTotalIdxWrite].uiSize	:= LEN(pa_tyXMLTable[iTotalIdxWrite].sValue);

	iTotalIdxWrite	:= iTotalIdxWrite + 1;

	pa_tyXMLTable[iTotalIdxWrite].sTitle	:= 'AT';
	pa_tyXMLTable[iTotalIdxWrite].sValue	:= 'Timestamp';
	pa_tyXMLTable[iTotalIdxWrite].uiSize	:= LEN(pa_tyXMLTable[iTotalIdxWrite].sValue);

	iTotalIdxWrite	:= iTotalIdxWrite + 1;

	pa_tyXMLTable[iTotalIdxWrite].sTitle	:= 'AV';
	pa_tyXMLTable[iTotalIdxWrite].sValue	:= sTimestamp;
	pa_tyXMLTable[iTotalIdxWrite].uiSize	:= LEN(pa_tyXMLTable[iTotalIdxWrite].sValue);

	iTotalIdxWrite	:= iTotalIdxWrite + 1;

	pa_tyXMLTable[iTotalIdxWrite].sTitle	:= 'EN';
	pa_tyXMLTable[iTotalIdxWrite].sValue	:= '';
	pa_tyXMLTable[iTotalIdxWrite].uiSize	:= LEN(pa_tyXMLTable[iTotalIdxWrite].sValue);

	iTotalIdxWrite	:= iTotalIdxWrite + 1;

	pa_tyXMLTable[iTotalIdxWrite].sTitle	:= 'ST';
	pa_tyXMLTable[iTotalIdxWrite].sValue	:= 'SendBoardInfo';
	pa_tyXMLTable[iTotalIdxWrite].uiSize	:= LEN(pa_tyXMLTable[iTotalIdxWrite].sValue);

	iTotalIdxWrite	:= iTotalIdxWrite + 1;

	IF tyParameter.tyAvl.bBoardId = TRUE THEN
		pa_tyXMLTable[iTotalIdxWrite].sTitle	:= 'AT';
		pa_tyXMLTable[iTotalIdxWrite].sValue	:= 'BoardId';
		pa_tyXMLTable[iTotalIdxWrite].uiSize	:= LEN(pa_tyXMLTable[iTotalIdxWrite].sValue);

		iTotalIdxWrite	:= iTotalIdxWrite + 1;

		pa_tyXMLTable[iTotalIdxWrite].sTitle	:= 'AV';
		pa_tyXMLTable[iTotalIdxWrite].sValue	:= tyParameter.tyData.sBoardId;
		pa_tyXMLTable[iTotalIdxWrite].uiSize	:= LEN(pa_tyXMLTable[iTotalIdxWrite].sValue);

		iTotalIdxWrite	:= iTotalIdxWrite + 1;
	END_IF

	IF tyParameter.tyAvl.bBoardIdCreatedBy = TRUE THEN
		pa_tyXMLTable[iTotalIdxWrite].sTitle	:= 'AT';
		pa_tyXMLTable[iTotalIdxWrite].sValue	:= 'BoardIdCreatedBy';
		pa_tyXMLTable[iTotalIdxWrite].uiSize	:= LEN(pa_tyXMLTable[iTotalIdxWrite].sValue);

		iTotalIdxWrite	:= iTotalIdxWrite + 1;

		pa_tyXMLTable[iTotalIdxWrite].sTitle	:= 'AV';
		pa_tyXMLTable[iTotalIdxWrite].sValue	:= tyParameter.tyData.sBoardIdCreatedBy;
		pa_tyXMLTable[iTotalIdxWrite].uiSize	:= LEN(pa_tyXMLTable[iTotalIdxWrite].sValue);

		iTotalIdxWrite	:= iTotalIdxWrite + 1;
	END_IF

	IF tyParameter.tyAvl.bFailedBoard = TRUE THEN
		pa_tyXMLTable[iTotalIdxWrite].sTitle	:= 'AT';
		pa_tyXMLTable[iTotalIdxWrite].sValue	:= 'FailedBoard';
		pa_tyXMLTable[iTotalIdxWrite].uiSize	:= LEN(pa_tyXMLTable[iTotalIdxWrite].sValue);

		iTotalIdxWrite	:= iTotalIdxWrite + 1;

		pa_tyXMLTable[iTotalIdxWrite].sTitle	:= 'AV';
		pa_tyXMLTable[iTotalIdxWrite].sValue	:= DINT_TO_STRING(UDINT_TO_DINT(tyParameter.tyData.eFailedBoard));
		pa_tyXMLTable[iTotalIdxWrite].uiSize	:= LEN(pa_tyXMLTable[iTotalIdxWrite].sValue);

		iTotalIdxWrite	:= iTotalIdxWrite + 1;
	END_IF

	IF tyParameter.tyAvl.bProductTypeId = TRUE THEN
		pa_tyXMLTable[iTotalIdxWrite].sTitle	:= 'AT';
		pa_tyXMLTable[iTotalIdxWrite].sValue	:= 'ProductTypeId';
		pa_tyXMLTable[iTotalIdxWrite].uiSize	:= LEN(pa_tyXMLTable[iTotalIdxWrite].sValue);

		iTotalIdxWrite	:= iTotalIdxWrite + 1;

		pa_tyXMLTable[iTotalIdxWrite].sTitle	:= 'AV';
		pa_tyXMLTable[iTotalIdxWrite].sValue	:= tyParameter.tyData.sProductTypeId;
		pa_tyXMLTable[iTotalIdxWrite].uiSize	:= LEN(pa_tyXMLTable[iTotalIdxWrite].sValue);

		iTotalIdxWrite	:= iTotalIdxWrite + 1;
	END_IF

	IF tyParameter.tyAvl.bFlippedBoard = TRUE THEN
		pa_tyXMLTable[iTotalIdxWrite].sTitle	:= 'AT';
		pa_tyXMLTable[iTotalIdxWrite].sValue	:= 'FlippedBoard';
		pa_tyXMLTable[iTotalIdxWrite].uiSize	:= LEN(pa_tyXMLTable[iTotalIdxWrite].sValue);

		iTotalIdxWrite	:= iTotalIdxWrite + 1;

		pa_tyXMLTable[iTotalIdxWrite].sTitle	:= 'AV';
		pa_tyXMLTable[iTotalIdxWrite].sValue	:= DINT_TO_STRING(UDINT_TO_DINT(tyParameter.tyData.eFlippedBoard));
		pa_tyXMLTable[iTotalIdxWrite].uiSize	:= LEN(pa_tyXMLTable[iTotalIdxWrite].sValue);

		iTotalIdxWrite	:= iTotalIdxWrite + 1;
	END_IF

	IF tyParameter.tyAvl.bTopBarcode = TRUE THEN
		pa_tyXMLTable[iTotalIdxWrite].sTitle	:= 'AT';
		pa_tyXMLTable[iTotalIdxWrite].sValue	:= 'TopBarcode';
		pa_tyXMLTable[iTotalIdxWrite].uiSize	:= LEN(pa_tyXMLTable[iTotalIdxWrite].sValue);

		iTotalIdxWrite	:= iTotalIdxWrite + 1;

		pa_tyXMLTable[iTotalIdxWrite].sTitle	:= 'AV';
		pa_tyXMLTable[iTotalIdxWrite].sValue	:= tyParameter.tyData.sTopBarcode;
		pa_tyXMLTable[iTotalIdxWrite].uiSize	:= LEN(pa_tyXMLTable[iTotalIdxWrite].sValue);

		iTotalIdxWrite	:= iTotalIdxWrite + 1;
	END_IF

	IF tyParameter.tyAvl.bBottomBarcode = TRUE THEN
		pa_tyXMLTable[iTotalIdxWrite].sTitle	:= 'AT';
		pa_tyXMLTable[iTotalIdxWrite].sValue	:= 'BottomBarcode';
		pa_tyXMLTable[iTotalIdxWrite].uiSize	:= LEN(pa_tyXMLTable[iTotalIdxWrite].sValue);

		iTotalIdxWrite	:= iTotalIdxWrite + 1;

		pa_tyXMLTable[iTotalIdxWrite].sTitle	:= 'AV';
		pa_tyXMLTable[iTotalIdxWrite].sValue	:= tyParameter.tyData.sBottomBarcode;
		pa_tyXMLTable[iTotalIdxWrite].uiSize	:= LEN(pa_tyXMLTable[iTotalIdxWrite].sValue);

		iTotalIdxWrite	:= iTotalIdxWrite + 1;
	END_IF

	IF tyParameter.tyAvl.bLength = TRUE THEN
		pa_tyXMLTable[iTotalIdxWrite].sTitle	:= 'AT';
		pa_tyXMLTable[iTotalIdxWrite].sValue	:= 'Length';
		pa_tyXMLTable[iTotalIdxWrite].uiSize	:= LEN(pa_tyXMLTable[iTotalIdxWrite].sValue);

		iTotalIdxWrite	:= iTotalIdxWrite + 1;

		pa_tyXMLTable[iTotalIdxWrite].sTitle	:= 'AV';
		pa_tyXMLTable[iTotalIdxWrite].sValue	:= REAL_TO_STRING(tyParameter.tyData.rLength);
		pa_tyXMLTable[iTotalIdxWrite].uiSize	:= LEN(pa_tyXMLTable[iTotalIdxWrite].sValue);

		iTotalIdxWrite	:= iTotalIdxWrite + 1;
	END_IF

	IF tyParameter.tyAvl.bWidth = TRUE THEN
		pa_tyXMLTable[iTotalIdxWrite].sTitle	:= 'AT';
		pa_tyXMLTable[iTotalIdxWrite].sValue	:= 'Width';
		pa_tyXMLTable[iTotalIdxWrite].uiSize	:= LEN(pa_tyXMLTable[iTotalIdxWrite].sValue);

		iTotalIdxWrite	:= iTotalIdxWrite + 1;

		pa_tyXMLTable[iTotalIdxWrite].sTitle	:= 'AV';
		pa_tyXMLTable[iTotalIdxWrite].sValue	:= REAL_TO_STRING(tyParameter.tyData.rWidth);
		pa_tyXMLTable[iTotalIdxWrite].uiSize	:= LEN(pa_tyXMLTable[iTotalIdxWrite].sValue);

		iTotalIdxWrite	:= iTotalIdxWrite + 1;
	END_IF

	IF tyParameter.tyAvl.bThickness = TRUE THEN
		pa_tyXMLTable[iTotalIdxWrite].sTitle	:= 'AT';
		pa_tyXMLTable[iTotalIdxWrite].sValue	:= 'Thickness';
		pa_tyXMLTable[iTotalIdxWrite].uiSize	:= LEN(pa_tyXMLTable[iTotalIdxWrite].sValue);

		iTotalIdxWrite	:= iTotalIdxWrite + 1;

		pa_tyXMLTable[iTotalIdxWrite].sTitle	:= 'AV';
		pa_tyXMLTable[iTotalIdxWrite].sValue	:= REAL_TO_STRING(tyParameter.tyData.rThickness);
		pa_tyXMLTable[iTotalIdxWrite].uiSize	:= LEN(pa_tyXMLTable[iTotalIdxWrite].sValue);

		iTotalIdxWrite	:= iTotalIdxWrite + 1;
	END_IF

	IF tyParameter.tyAvl.bTopClearanceHeight = TRUE THEN
		pa_tyXMLTable[iTotalIdxWrite].sTitle	:= 'AT';
		pa_tyXMLTable[iTotalIdxWrite].sValue	:= 'TopClearanceHeight';
		pa_tyXMLTable[iTotalIdxWrite].uiSize	:= LEN(pa_tyXMLTable[iTotalIdxWrite].sValue);

		iTotalIdxWrite	:= iTotalIdxWrite + 1;

		pa_tyXMLTable[iTotalIdxWrite].sTitle	:= 'AV';
		pa_tyXMLTable[iTotalIdxWrite].sValue	:= REAL_TO_STRING(tyParameter.tyData.rTopClearanceHeight);
		pa_tyXMLTable[iTotalIdxWrite].uiSize	:= LEN(pa_tyXMLTable[iTotalIdxWrite].sValue);

		iTotalIdxWrite	:= iTotalIdxWrite + 1;
	END_IF

	IF tyParameter.tyAvl.bBottomClearanceHeight = TRUE THEN
		pa_tyXMLTable[iTotalIdxWrite].sTitle	:= 'AT';
		pa_tyXMLTable[iTotalIdxWrite].sValue	:= 'BottomClearanceHeight';
		pa_tyXMLTable[iTotalIdxWrite].uiSize	:= LEN(pa_tyXMLTable[iTotalIdxWrite].sValue);

		iTotalIdxWrite	:= iTotalIdxWrite + 1;

		pa_tyXMLTable[iTotalIdxWrite].sTitle	:= 'AV';
		pa_tyXMLTable[iTotalIdxWrite].sValue	:= REAL_TO_STRING(tyParameter.tyData.rBottomClearanceHeight);
		pa_tyXMLTable[iTotalIdxWrite].uiSize	:= LEN(pa_tyXMLTable[iTotalIdxWrite].sValue);

		iTotalIdxWrite	:= iTotalIdxWrite + 1;
	END_IF

	IF tyParameter.tyAvl.bWeight = TRUE THEN
		pa_tyXMLTable[iTotalIdxWrite].sTitle	:= 'AT';
		pa_tyXMLTable[iTotalIdxWrite].sValue	:= 'Weight';
		pa_tyXMLTable[iTotalIdxWrite].uiSize	:= LEN(pa_tyXMLTable[iTotalIdxWrite].sValue);

		iTotalIdxWrite	:= iTotalIdxWrite + 1;

		pa_tyXMLTable[iTotalIdxWrite].sTitle	:= 'AV';
		pa_tyXMLTable[iTotalIdxWrite].sValue	:= REAL_TO_STRING(tyParameter.tyData.rWeight);
		pa_tyXMLTable[iTotalIdxWrite].uiSize	:= LEN(pa_tyXMLTable[iTotalIdxWrite].sValue);

		iTotalIdxWrite	:= iTotalIdxWrite + 1;
	END_IF

	IF tyParameter.tyAvl.bWorkOrderId = TRUE THEN
		pa_tyXMLTable[iTotalIdxWrite].sTitle	:= 'AT';
		pa_tyXMLTable[iTotalIdxWrite].sValue	:= 'WorkOrderId';
		pa_tyXMLTable[iTotalIdxWrite].uiSize	:= LEN(pa_tyXMLTable[iTotalIdxWrite].sValue);

		iTotalIdxWrite	:= iTotalIdxWrite + 1;

		pa_tyXMLTable[iTotalIdxWrite].sTitle	:= 'AV';
		pa_tyXMLTable[iTotalIdxWrite].sValue	:= tyParameter.tyData.sWorkOrderId;
		pa_tyXMLTable[iTotalIdxWrite].uiSize	:= LEN(pa_tyXMLTable[iTotalIdxWrite].sValue);

		iTotalIdxWrite	:= iTotalIdxWrite + 1;
	END_IF

	IF tyParameter.tyAvl.bBatchId = TRUE THEN
		pa_tyXMLTable[iTotalIdxWrite].sTitle	:= 'AT';
		pa_tyXMLTable[iTotalIdxWrite].sValue	:= 'BatchId';
		pa_tyXMLTable[iTotalIdxWrite].uiSize	:= LEN(pa_tyXMLTable[iTotalIdxWrite].sValue);

		iTotalIdxWrite	:= iTotalIdxWrite + 1;

		pa_tyXMLTable[iTotalIdxWrite].sTitle	:= 'AV';
		pa_tyXMLTable[iTotalIdxWrite].sValue	:= tyParameter.tyData.sBatchId;
		pa_tyXMLTable[iTotalIdxWrite].uiSize	:= LEN(pa_tyXMLTable[iTotalIdxWrite].sValue);

		iTotalIdxWrite	:= iTotalIdxWrite + 1;
	END_IF

	pa_tyXMLTable[iTotalIdxWrite].sTitle	:= 'ES';
	pa_tyXMLTable[iTotalIdxWrite].sValue	:= '';
	pa_tyXMLTable[iTotalIdxWrite].uiSize	:= LEN(pa_tyXMLTable[iTotalIdxWrite].sValue);

	iTotalIdxWrite	:= iTotalIdxWrite + 1;

	pa_tyXMLTable[iTotalIdxWrite].sTitle	:= 'ET';
	pa_tyXMLTable[iTotalIdxWrite].sValue	:= 'Hermes';
	pa_tyXMLTable[iTotalIdxWrite].uiSize	:= LEN(pa_tyXMLTable[iTotalIdxWrite].sValue);

	iTotalIdxWrite	:= iTotalIdxWrite + 1;

	pa_tyXMLTable[iTotalIdxWrite].sTitle	:= 'EN';
	pa_tyXMLTable[iTotalIdxWrite].sValue	:= '';
	pa_tyXMLTable[iTotalIdxWrite].uiSize	:= LEN(pa_tyXMLTable[iTotalIdxWrite].sValue);

	iTotalIdxWrite	:= iTotalIdxWrite + 1;

	iTotalIdxWrite	:= fHermesFormSendBoardInfo;

END_FUNCTION
```
